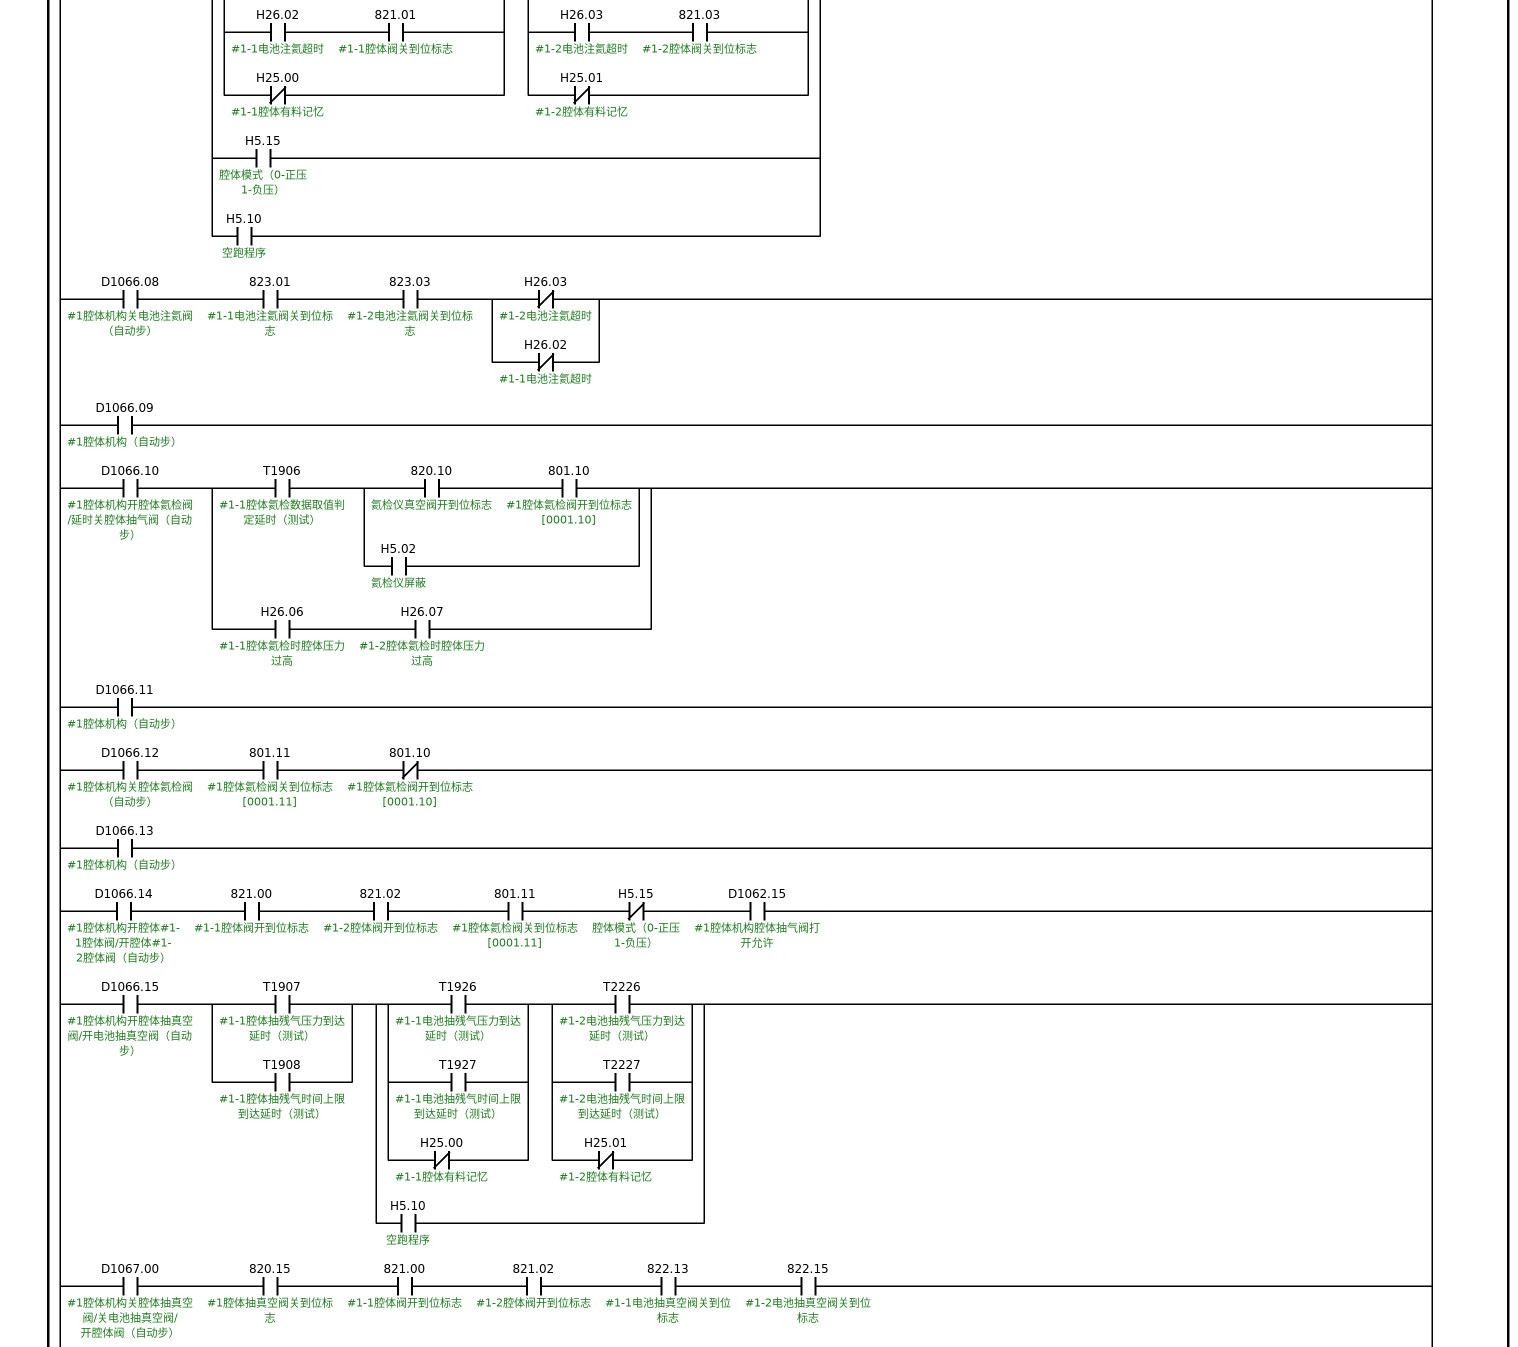
; [picture p192: 氦检机构 / 氦检腔1自动, rungs 7-7]

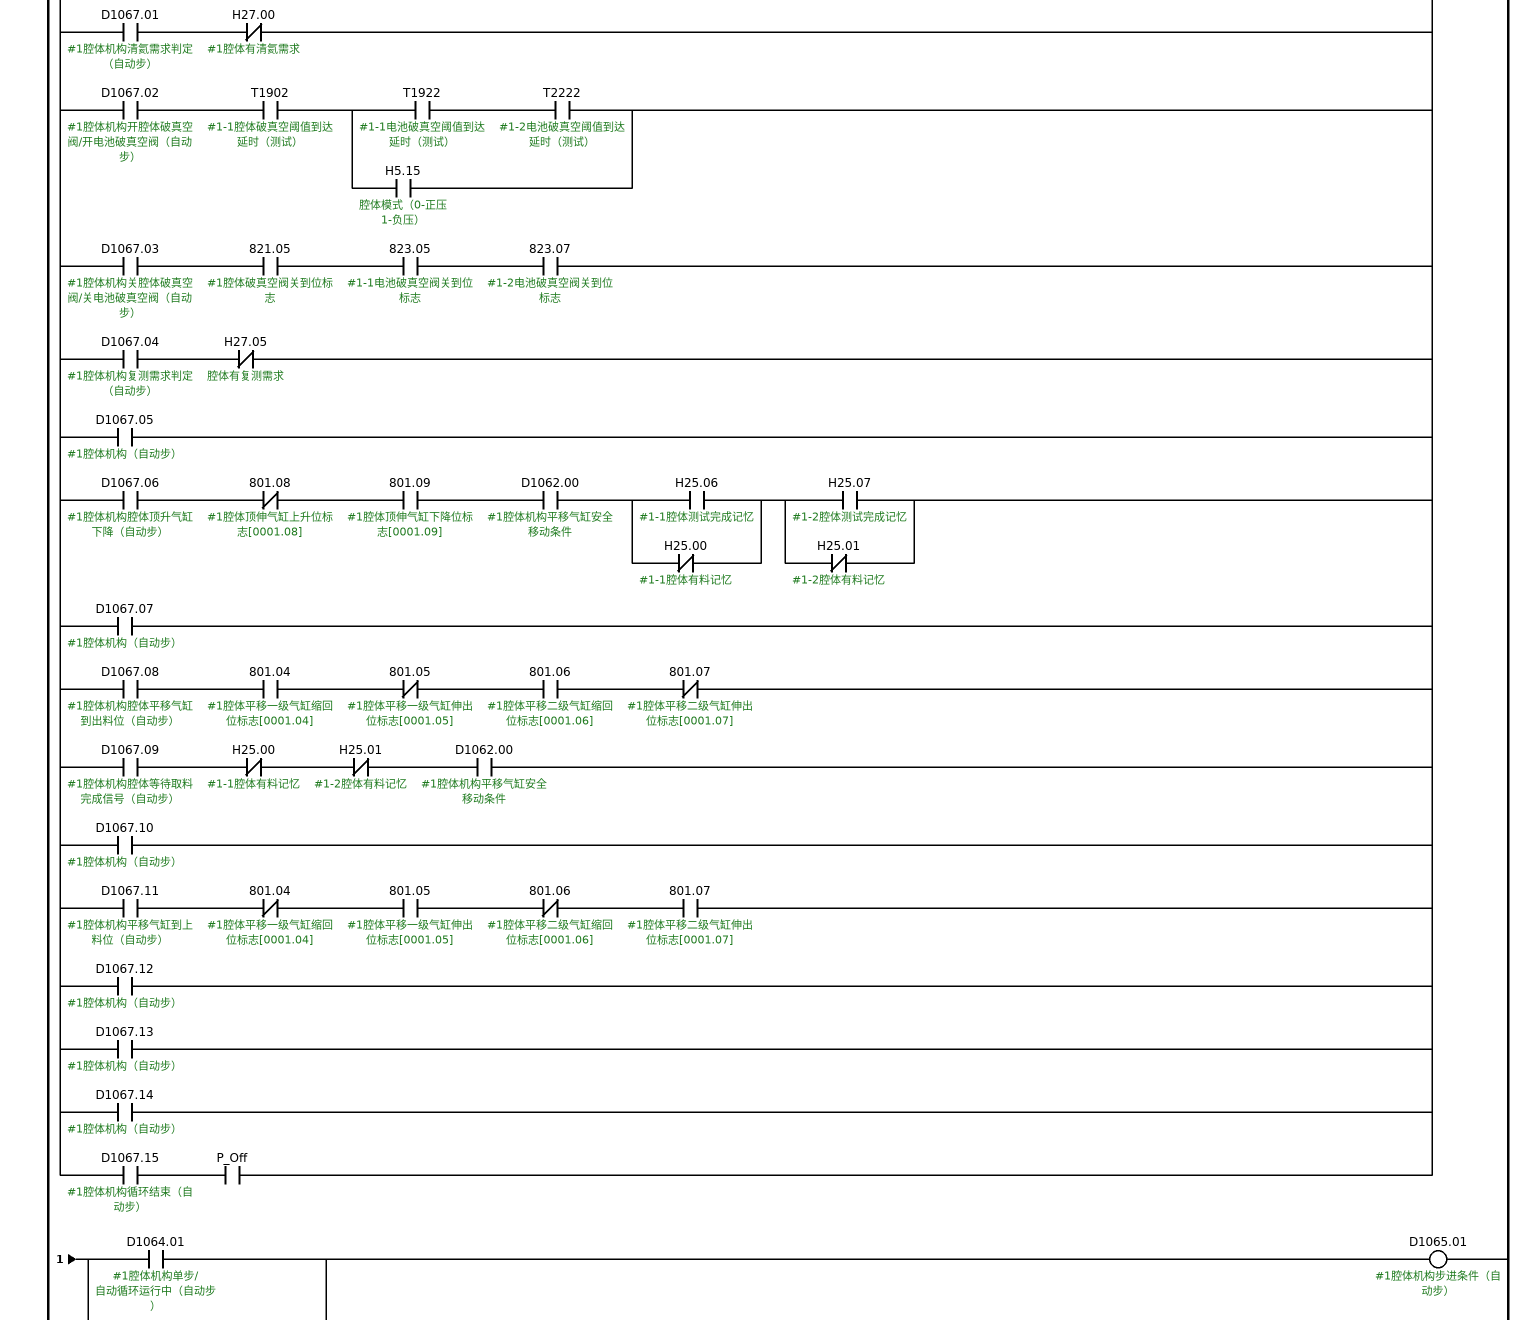

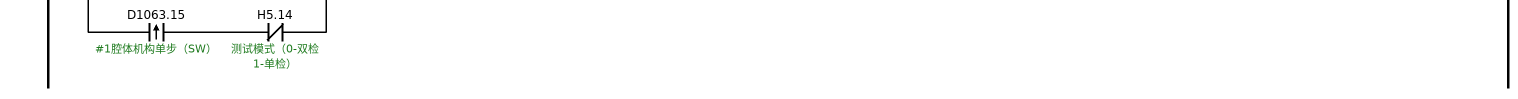
; rung 7: #1腔体机构步进条件（自动步）
LD D1066.00  ; #1腔体机构自动开始（自动步）
AND T1530  ; #1腔体机构开始运行条件延时(自动步)
LD D1066.01  ; #1腔体机构平移气缸到氦检位/数据初始化（自动步）
ANDNOT 801.04  ; #1腔体平移一级气缸缩回位标志[0001.04]
AND 801.05  ; #1腔体平移一级气缸伸出位标志[0001.05]
AND 801.06  ; #1腔体平移二级气缸缩回位标志[0001.06]
ANDNOT 801.07  ; #1腔体平移二级气缸伸出位标志[0001.07]
AND T1531  ; #1腔体机构数据初始化延时（自动步）
ORLD
LD D1066.02  ; #1腔体机构腔体顶升气缸上升（自动步）
AND 801.08  ; #1腔体顶伸气缸上升位标志[0001.08]
ANDNOT 801.09  ; #1腔体顶伸气缸下降位标志[0001.09]
ORLD
LD D1066.03  ; #1腔体机构等待氦检阀打开条件及腔体抽气阀打开条件/开腔体阀（自动步）
AND 821.00  ; #1-1腔体阀开到位标志
AND 821.02  ; #1-2腔体阀开到位标志
ANDNOT H32.00  ; #2腔体有清氦需求
ANDNOT H37.00  ; #3腔体有清氦需求
AND D1062.15  ; #1腔体机构腔体抽气阀打开允许
AND D1062.14  ; #1腔体氦检阀打开允许条件
LD W380.15  ; 氦检仪漏率低于设定值（稳态）
OR H5.02  ; 氦检仪屏蔽
ANDLD
AND=L(301) D1074 #0  ; #1腔体机构清氦步序号
ORLD
OR D1066.04  ; #1腔体机构（自动步）
LD D1066.05  ; #1腔体机构腔体抽气阀打开/延时开电池抽气阀（自动步）
LD T1900  ; #1-1腔体抽真空阈值到达延时（测试）
LD 822.12  ; #1-1电池抽真空阀开到位标志
AND T1920  ; #1-1电池抽真空阈值到达延时（测试）
LD H26.00  ; #1-1电池泄漏
ANDNOT H26.01  ; #1-2电池泄漏
ORLD
ORNOT H25.00  ; #1-1腔体有料记忆
LD 822.14  ; #1-2电池抽真空阀开到位标志
AND T2220  ; #1-2电池抽真空阈值到达延时（测试）
LDNOT H26.00  ; #1-1电池泄漏
AND H26.01  ; #1-2电池泄漏
ORLD
ORNOT H25.01  ; #1-2腔体有料记忆
ANDLD
OR H5.15  ; 腔体模式（0-正压 1-负压）
OR H5.10  ; 空跑程序
ANDLD
LD H26.04  ; #1-1腔体抽真空NG
ORNOT H25.00  ; #1-1腔体有料记忆
LD H26.05  ; #1-2腔体抽真空NG
ORNOT H25.01  ; #1-2腔体有料记忆
ANDLD
ORLD
LD H26.00  ; #1-1电池泄漏
AND H26.01  ; #1-2电池泄漏
ORLD
ANDLD
ORLD
LD D1066.06  ; #1腔体机构关电池抽气阀（自动步）  // 单个电池出现电池泄漏时，需将对应的腔体阀门关闭
ANDNOT W407.14  ; 设备氦气压力信号[alm]
ANDNOT W407.15  ; 精密调压阀信号[alm]
AND 822.13  ; #1-1电池抽真空阀关到位标志
AND 822.15  ; #1-2电池抽真空阀关到位标志
ANDNOT H26.04  ; #1-1腔体抽真空NG
ANDNOT H26.05  ; #1-2腔体抽真空NG
LD H26.00  ; #1-1电池泄漏
AND 821.01  ; #1-1腔体阀关到位标志
ORNOT H26.00  ; #1-1电池泄漏
ORNOT H25.00  ; #1-1腔体有料记忆
ANDLD
LD H26.01  ; #1-2电池泄漏
AND 821.03  ; #1-2腔体阀关到位标志
ORNOT H26.01  ; #1-2电池泄漏
ORNOT H25.01  ; #1-2腔体有料记忆
ANDLD
ORLD
LD D1066.07  ; #1腔体机构开电池注氦阀（自动步）  // 单个电池出现注氦超时时，需将对应的腔体阀门关闭
LD 823.00  ; #1-1电池注氦阀开到位标志
AND T1924  ; #1-1电池注氦压力到达延时（测试）
OR H26.00  ; #1-1电池泄漏
LD H26.02  ; #1-1电池注氦超时
AND 821.01  ; #1-1腔体阀关到位标志
ORLD
ORNOT H25.00  ; #1-1腔体有料记忆
LD 823.02  ; #1-2电池注氦阀开到位标志
AND T2224  ; #1-2电池注氦压力到达延时（测试）
OR H26.01  ; #1-2电池泄漏
LD H26.03  ; #1-2电池注氦超时
AND 821.03  ; #1-2腔体阀关到位标志
ORLD
ORNOT H25.01  ; #1-2腔体有料记忆
ANDLD
OR H5.15  ; 腔体模式（0-正压 1-负压）
OR H5.10  ; 空跑程序
ANDLD
ORLD
LD D1066.08  ; #1腔体机构关电池注氦阀（自动步）
AND 823.01  ; #1-1电池注氦阀关到位标志
AND 823.03  ; #1-2电池注氦阀关到位标志
LDNOT H26.03  ; #1-2电池注氦超时
ORNOT H26.02  ; #1-1电池注氦超时
ANDLD
ORLD
OR D1066.09  ; #1腔体机构（自动步）
LD D1066.10  ; #1腔体机构开腔体氦检阀/延时关腔体抽气阀（自动步）
LD T1906  ; #1-1腔体氦检数据取值判定延时（测试）
LD 820.10  ; 氦检仪真空阀开到位标志
AND 801.10  ; #1腔体氦检阀开到位标志[0001.10]
OR H5.02  ; 氦检仪屏蔽
ANDLD
LD H26.06  ; #1-1腔体氦检时腔体压力过高
AND H26.07  ; #1-2腔体氦检时腔体压力过高
ORLD
ANDLD
ORLD
OR D1066.11  ; #1腔体机构（自动步）
LD D1066.12  ; #1腔体机构关腔体氦检阀（自动步）
AND 801.11  ; #1腔体氦检阀关到位标志[0001.11]
ANDNOT 801.10  ; #1腔体氦检阀开到位标志[0001.10]
ORLD
OR D1066.13  ; #1腔体机构（自动步）
LD D1066.14  ; #1腔体机构开腔体#1-1腔体阀/开腔体#1-2腔体阀（自动步）
AND 821.00  ; #1-1腔体阀开到位标志
AND 821.02  ; #1-2腔体阀开到位标志
AND 801.11  ; #1腔体氦检阀关到位标志[0001.11]
ANDNOT H5.15  ; 腔体模式（0-正压 1-负压）
AND D1062.15  ; #1腔体机构腔体抽气阀打开允许
ORLD
LD D1066.15  ; #1腔体机构开腔体抽真空阀/开电池抽真空阀（自动步）
LD T1907  ; #1-1腔体抽残气压力到达延时（测试）
OR T1908  ; #1-1腔体抽残气时间上限到达延时（测试）
ANDLD
LD T1926  ; #1-1电池抽残气压力到达延时（测试）
OR T1927  ; #1-1电池抽残气时间上限到达延时（测试）
ORNOT H25.00  ; #1-1腔体有料记忆
LD T2226  ; #1-2电池抽残气压力到达延时（测试）
OR T2227  ; #1-2电池抽残气时间上限到达延时（测试）
ORNOT H25.01  ; #1-2腔体有料记忆
ANDLD
OR H5.10  ; 空跑程序
ANDLD
ORLD
LD D1067.00  ; #1腔体机构关腔体抽真空阀/关电池抽真空阀/开腔体阀（自动步）
AND 820.15  ; #1腔体抽真空阀关到位标志
AND 821.00  ; #1-1腔体阀开到位标志
AND 821.02  ; #1-2腔体阀开到位标志
AND 822.13  ; #1-1电池抽真空阀关到位标志
AND 822.15  ; #1-2电池抽真空阀关到位标志
ORLD
LD D1067.01  ; #1腔体机构清氦需求判定（自动步）
ANDNOT H27.00  ; #1腔体有清氦需求
ORLD
LD D1067.02  ; #1腔体机构开腔体破真空阀/开电池破真空阀（自动步）
AND T1902  ; #1-1腔体破真空阈值到达延时（测试）
LD T1922  ; #1-1电池破真空阈值到达延时（测试）
AND T2222  ; #1-2电池破真空阈值到达延时（测试）
OR H5.15  ; 腔体模式（0-正压 1-负压）
ANDLD
ORLD
LD D1067.03  ; #1腔体机构关腔体破真空阀/关电池破真空阀（自动步）
AND 821.05  ; #1腔体破真空阀关到位标志
AND 823.05  ; #1-1电池破真空阀关到位标志
AND 823.07  ; #1-2电池破真空阀关到位标志
ORLD
LD D1067.04  ; #1腔体机构复测需求判定（自动步）
ANDNOT H27.05  ; 腔体有复测需求
ORLD
OR D1067.05  ; #1腔体机构（自动步）
LD D1067.06  ; #1腔体机构腔体顶升气缸下降（自动步）
ANDNOT 801.08  ; #1腔体顶伸气缸上升位标志[0001.08]
AND 801.09  ; #1腔体顶伸气缸下降位标志[0001.09]
AND D1062.00  ; #1腔体机构平移气缸安全移动条件
LD H25.06  ; #1-1腔体测试完成记忆
ORNOT H25.00  ; #1-1腔体有料记忆
ANDLD
LD H25.07  ; #1-2腔体测试完成记忆
ORNOT H25.01  ; #1-2腔体有料记忆
ANDLD
ORLD
OR D1067.07  ; #1腔体机构（自动步）
LD D1067.08  ; #1腔体机构腔体平移气缸到出料位（自动步）
AND 801.04  ; #1腔体平移一级气缸缩回位标志[0001.04]
ANDNOT 801.05  ; #1腔体平移一级气缸伸出位标志[0001.05]
AND 801.06  ; #1腔体平移二级气缸缩回位标志[0001.06]
ANDNOT 801.07  ; #1腔体平移二级气缸伸出位标志[0001.07]
ORLD
LD D1067.09  ; #1腔体机构腔体等待取料完成信号（自动步）
ANDNOT H25.00  ; #1-1腔体有料记忆
ANDNOT H25.01  ; #1-2腔体有料记忆
AND D1062.00  ; #1腔体机构平移气缸安全移动条件
ORLD
OR D1067.10  ; #1腔体机构（自动步）
LD D1067.11  ; #1腔体机构平移气缸到上料位（自动步）
ANDNOT 801.04  ; #1腔体平移一级气缸缩回位标志[0001.04]
AND 801.05  ; #1腔体平移一级气缸伸出位标志[0001.05]
ANDNOT 801.06  ; #1腔体平移二级气缸缩回位标志[0001.06]
AND 801.07  ; #1腔体平移二级气缸伸出位标志[0001.07]
ORLD
OR D1067.12  ; #1腔体机构（自动步）
OR D1067.13  ; #1腔体机构（自动步）
OR D1067.14  ; #1腔体机构（自动步）
LD D1067.15  ; #1腔体机构循环结束（自动步）
AND P_Off
ORLD
LD D1064.01  ; #1腔体机构单步/自动循环运行中（自动步）
@LD D1063.15  ; #1腔体机构单步（SW）
ANDNOT H5.14  ; 测试模式（0-双检 1-单检）
ORLD
ANDLD
OUT D1065.01  ; #1腔体机构步进条件（自动步）

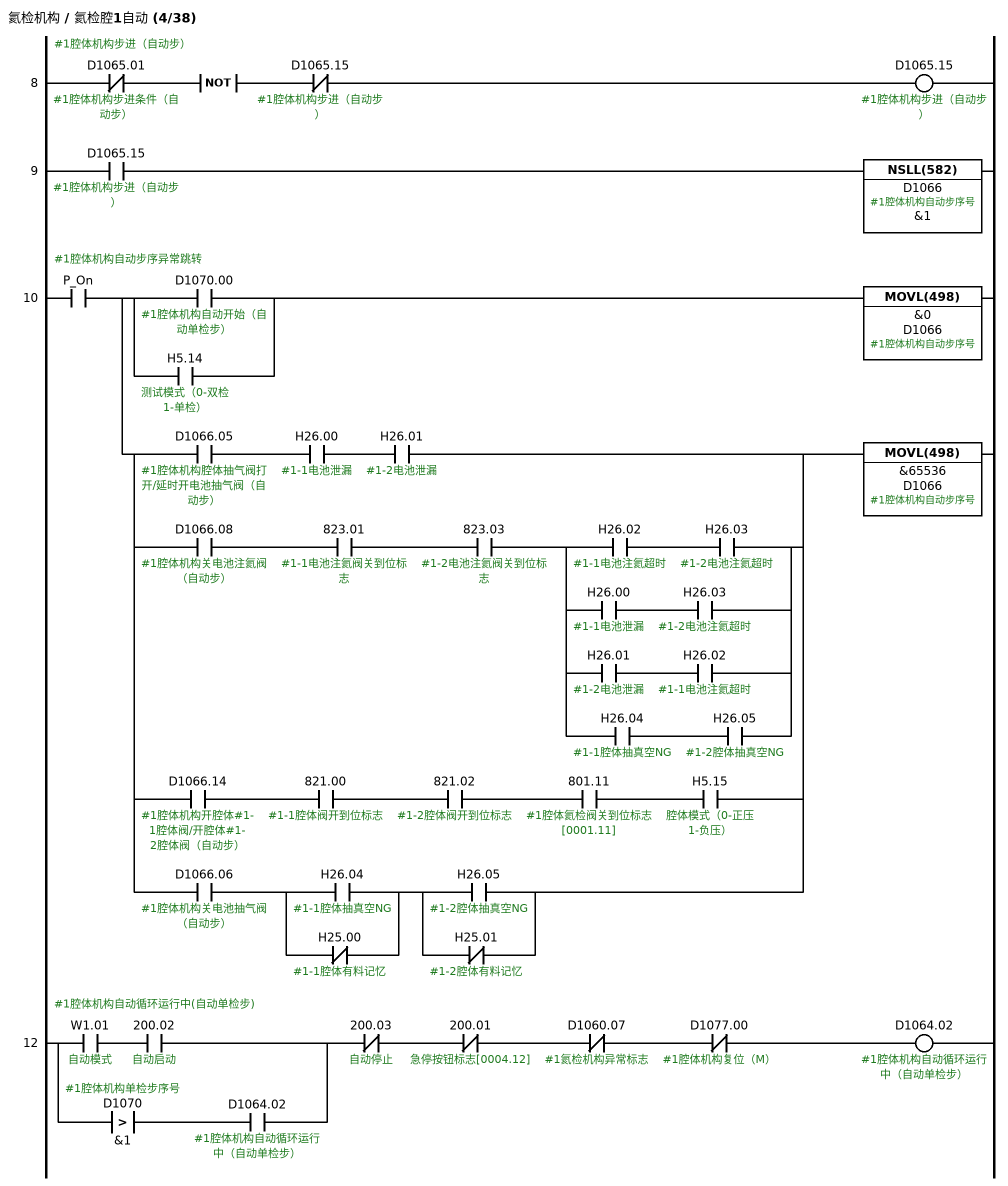
; rung 8: #1腔体机构步进（自动步）
LDNOT D1065.01  ; #1腔体机构步进条件（自动步）
NOT(520)
ANDNOT D1065.15  ; #1腔体机构步进（自动步）
OUT D1065.15  ; #1腔体机构步进（自动步）
; rung 9
LD D1065.15  ; #1腔体机构步进（自动步）
NSLL(582) D1066 &1  ; #1腔体机构自动步序号
; rung 10: #1腔体机构自动步序异常跳转
LD P_On
OUT TR0
LD D1070.00  ; #1腔体机构自动开始（自动单检步）
OR H5.14  ; 测试模式（0-双检 1-单检）
ANDLD
MOVL(498) &0 D1066  ; #1腔体机构自动步序号  // 测试模式为单检模式，腔体进入到复测步序时，将腔体机构自动步序清零
LD TR0
LD D1066.05  ; #1腔体机构腔体抽气阀打开/延时开电池抽气阀（自动步）
AND H26.00  ; #1-1电池泄漏
AND H26.01  ; #1-2电池泄漏
LD D1066.08  ; #1腔体机构关电池注氦阀（自动步）
AND 823.01  ; #1-1电池注氦阀关到位标志
AND 823.03  ; #1-2电池注氦阀关到位标志
LD H26.02  ; #1-1电池注氦超时
AND H26.03  ; #1-2电池注氦超时
LD H26.00  ; #1-1电池泄漏
AND H26.03  ; #1-2电池注氦超时
ORLD
LD H26.01  ; #1-2电池泄漏
AND H26.02  ; #1-1电池注氦超时
ORLD
LD H26.04  ; #1-1腔体抽真空NG
AND H26.05  ; #1-2腔体抽真空NG
ORLD
ANDLD
ORLD
LD D1066.14  ; #1腔体机构开腔体#1-1腔体阀/开腔体#1-2腔体阀（自动步）  // 负压模式不需要进行氦检后抽真空动作
AND 821.00  ; #1-1腔体阀开到位标志
AND 821.02  ; #1-2腔体阀开到位标志
AND 801.11  ; #1腔体氦检阀关到位标志[0001.11]
AND H5.15  ; 腔体模式（0-正压 1-负压）
ORLD
LD D1066.06  ; #1腔体机构关电池抽气阀（自动步）
LD H26.04  ; #1-1腔体抽真空NG
ORNOT H25.00  ; #1-1腔体有料记忆
ANDLD
LD H26.05  ; #1-2腔体抽真空NG
ORNOT H25.01  ; #1-2腔体有料记忆
ANDLD
ORLD
ANDLD
MOVL(498) &65536 D1066  ; #1腔体机构自动步序号  // 出现腔体抽真空NG，双电池抽真空NG，双电池注氦超时的情况，均跳转至自动步序D1067.0
; rung 11: ******************************* / 自动单检步序 / *******************************
; rung 12: #1腔体机构自动循环运行中(自动单检步)
LD W1.01  ; 自动模式
AND 200.02  ; 自动启动
LD>L(321) D1070 &1  ; #1腔体机构单检步序号
AND D1064.02  ; #1腔体机构自动循环运行中（自动单检步）
ORLD
ANDNOT 200.03  ; 自动停止
ANDNOT 200.01  ; 急停按钮标志[0004.12]
ANDNOT D1060.07  ; #1氦检机构异常标志
ANDNOT D1077.00  ; #1腔体机构复位（M）
OUT D1064.02  ; #1腔体机构自动循环运行中（自动单检步）

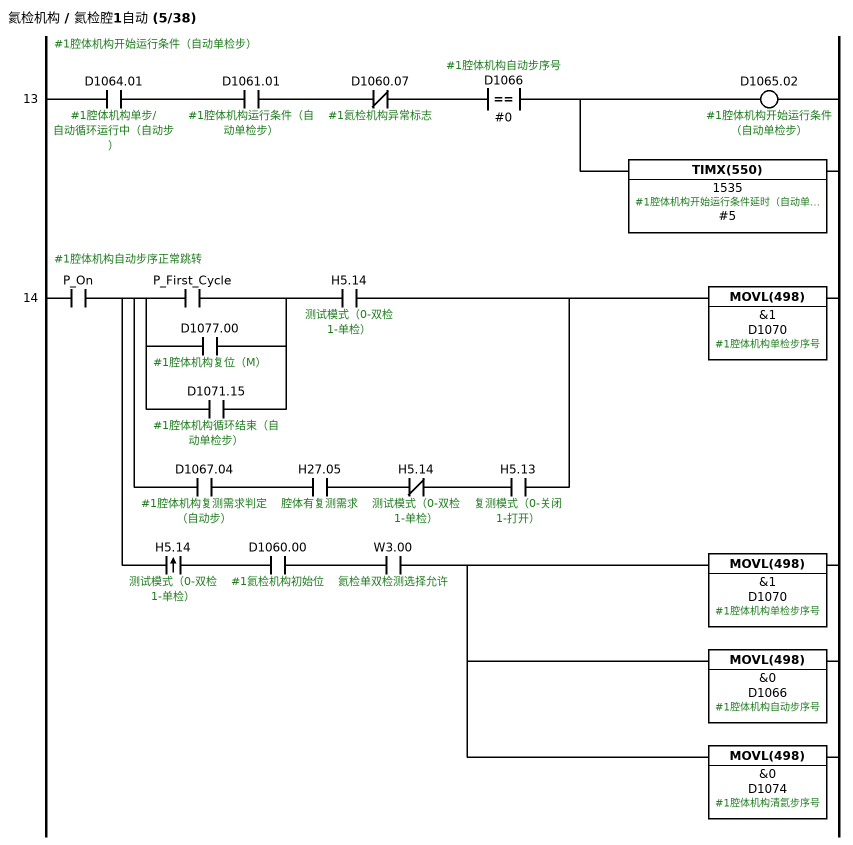
; rung 13: #1腔体机构开始运行条件（自动单检步）
LD D1064.01  ; #1腔体机构单步/自动循环运行中（自动步）
AND D1061.01  ; #1腔体机构运行条件（自动单检步）
ANDNOT D1060.07  ; #1氦检机构异常标志
AND=L(301) D1066 #0  ; #1腔体机构自动步序号
OUT D1065.02  ; #1腔体机构开始运行条件（自动单检步）
TIMX(550) 1535 #5  ; #1腔体机构开始运行条件延时（自动单检步）
; rung 14: #1腔体机构自动步序正常跳转
LD P_On
OUT TR0
LD P_First_Cycle
OR D1077.00  ; #1腔体机构复位（M）
OR D1071.15  ; #1腔体机构循环结束（自动单检步）
AND H5.14  ; 测试模式（0-双检 1-单检）
LD D1067.04  ; #1腔体机构复测需求判定（自动步）
AND H27.05  ; 腔体有复测需求
ANDNOT H5.14  ; 测试模式（0-双检 1-单检）
AND H5.13  ; 复测模式（0-关闭 1-打开）
ORLD
ANDLD
MOVL(498) &1 D1070  ; #1腔体机构单检步序号
LD TR0
@AND H5.14  ; 测试模式（0-双检 1-单检）
AND D1060.00  ; #1氦检机构初始位
AND W3.00  ; 氦检单双检测选择允许
MOVL(498) &1 D1070  ; #1腔体机构单检步序号
MOVL(498) &0 D1066  ; #1腔体机构自动步序号
MOVL(498) &0 D1074  ; #1腔体机构清氦步序号

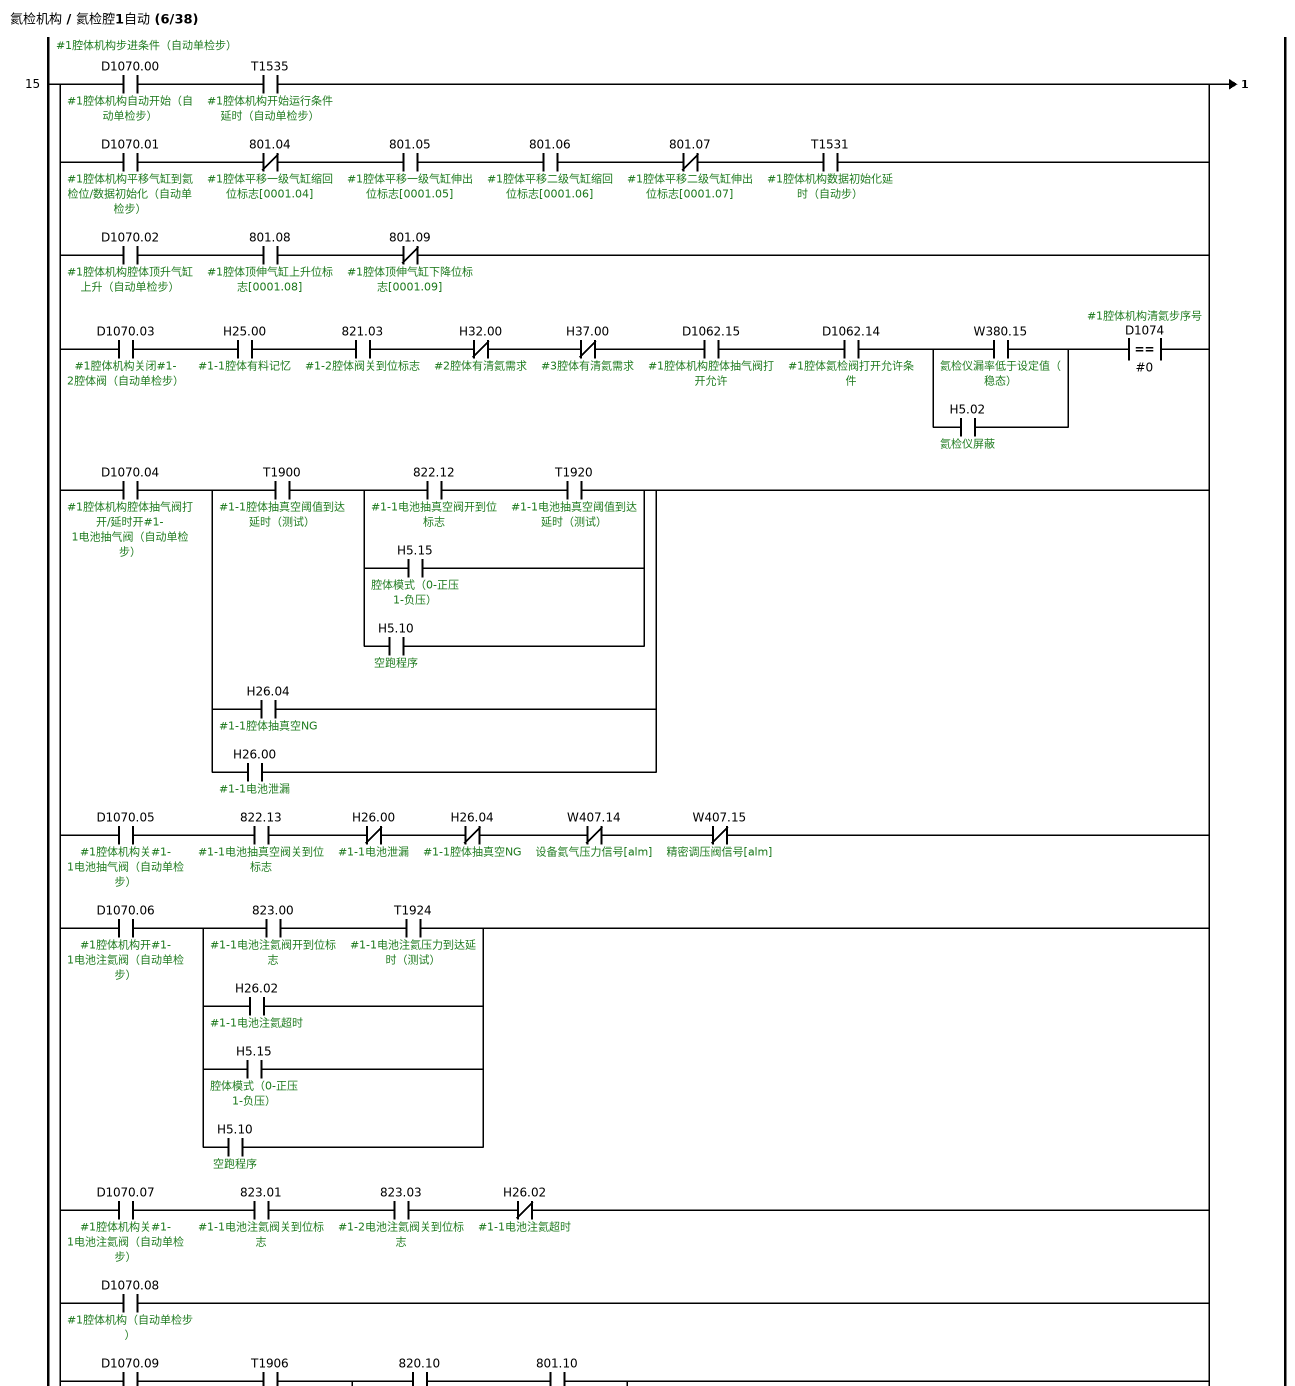

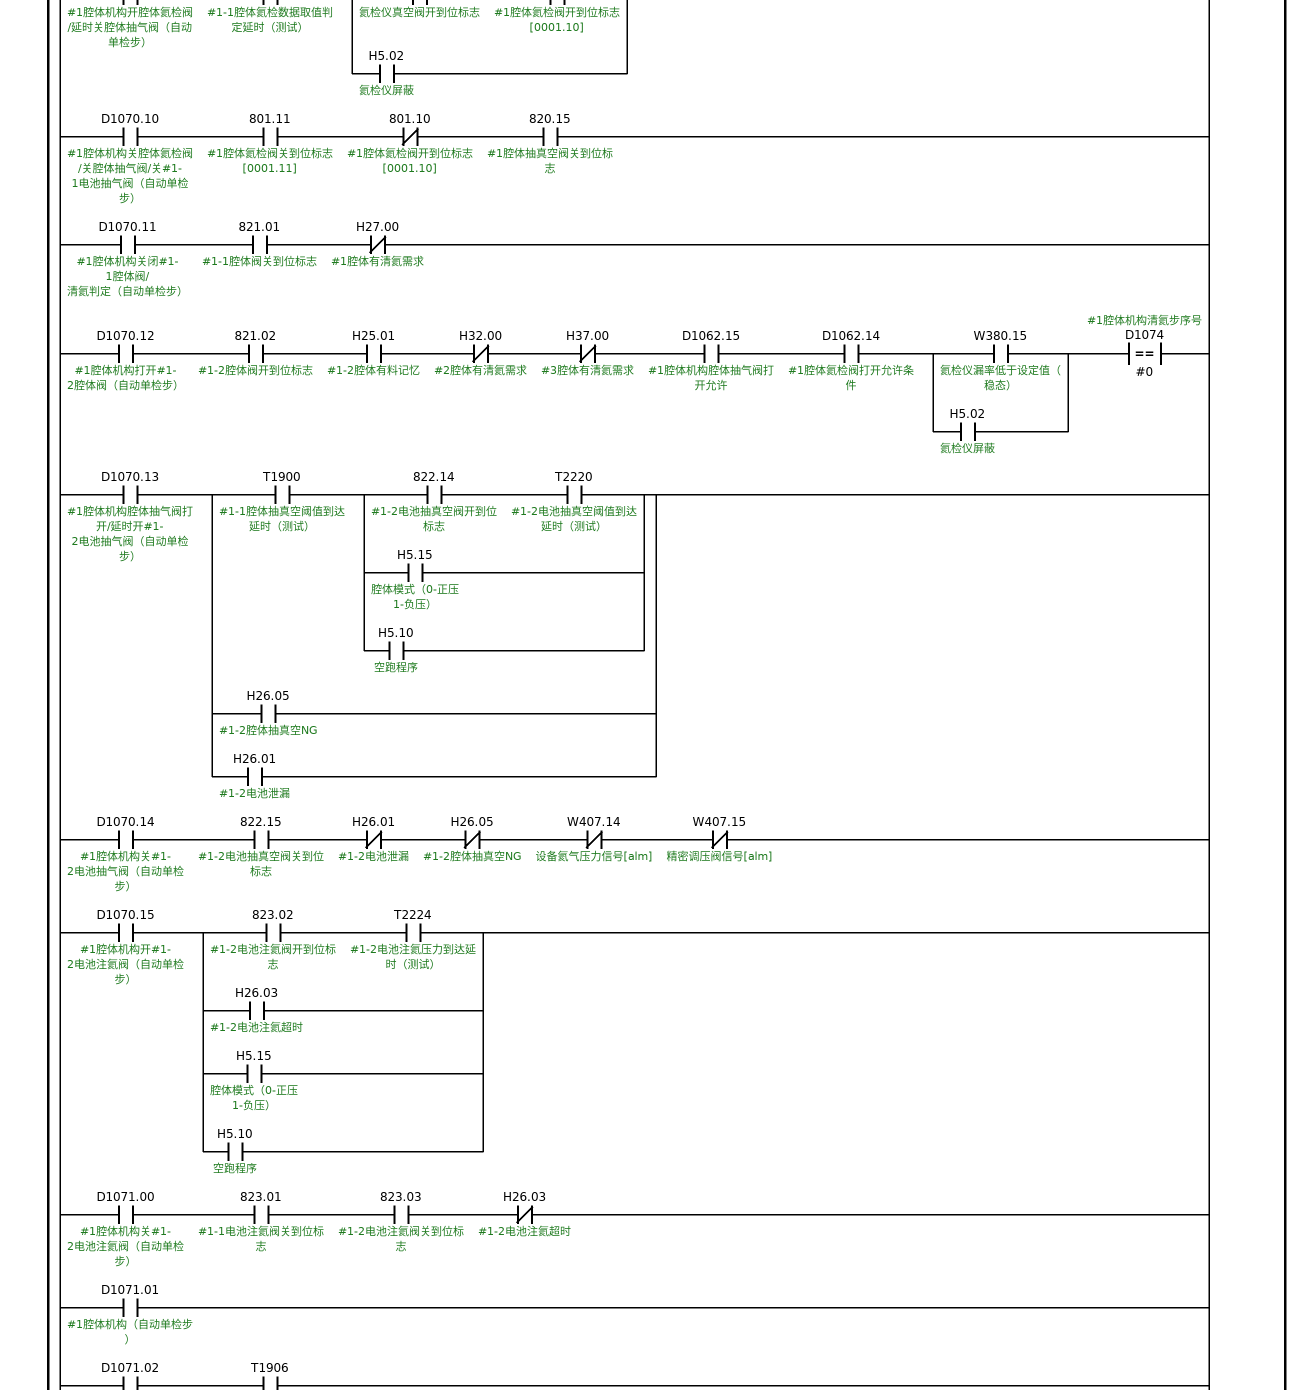

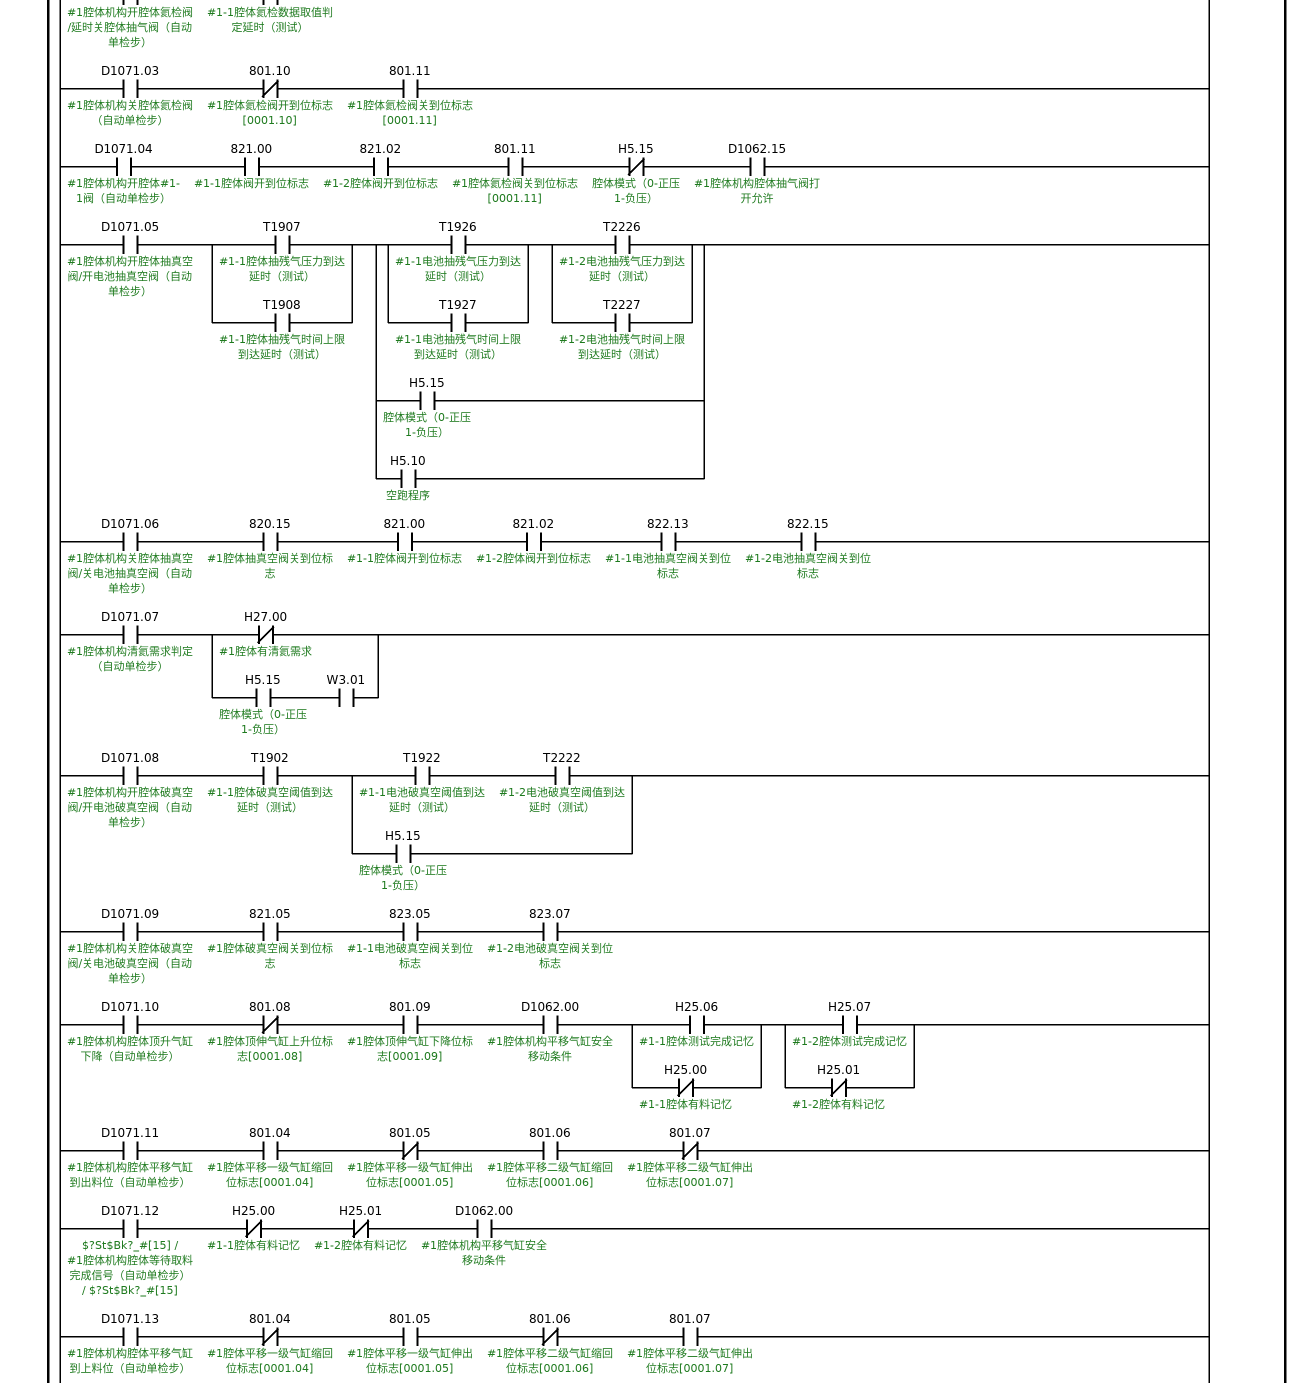

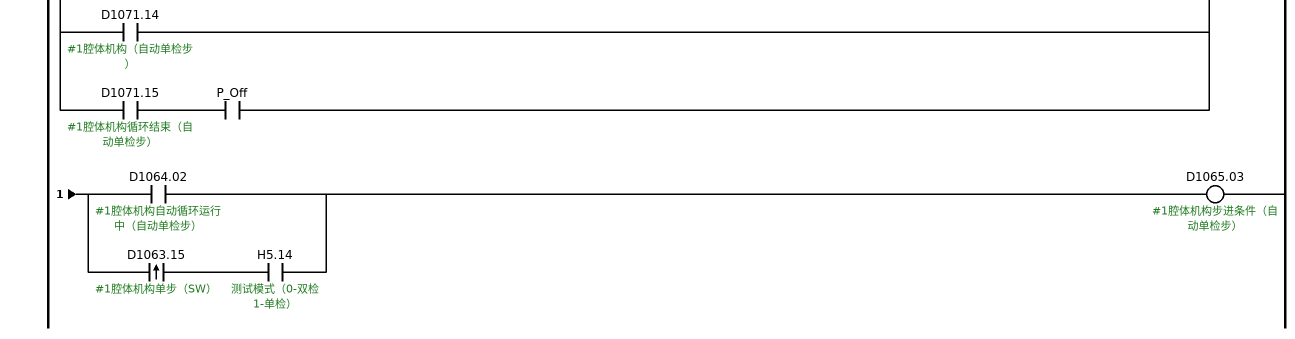
; rung 15: #1腔体机构步进条件（自动单检步）
LD D1070.00  ; #1腔体机构自动开始（自动单检步）
AND T1535  ; #1腔体机构开始运行条件延时（自动单检步）
LD D1070.01  ; #1腔体机构平移气缸到氦检位/数据初始化（自动单检步）
ANDNOT 801.04  ; #1腔体平移一级气缸缩回位标志[0001.04]
AND 801.05  ; #1腔体平移一级气缸伸出位标志[0001.05]
AND 801.06  ; #1腔体平移二级气缸缩回位标志[0001.06]
ANDNOT 801.07  ; #1腔体平移二级气缸伸出位标志[0001.07]
AND T1531  ; #1腔体机构数据初始化延时（自动步）
ORLD
LD D1070.02  ; #1腔体机构腔体顶升气缸上升（自动单检步）
AND 801.08  ; #1腔体顶伸气缸上升位标志[0001.08]
ANDNOT 801.09  ; #1腔体顶伸气缸下降位标志[0001.09]
ORLD
LD D1070.03  ; #1腔体机构关闭#1-2腔体阀（自动单检步）
AND H25.00  ; #1-1腔体有料记忆
AND 821.03  ; #1-2腔体阀关到位标志
ANDNOT H32.00  ; #2腔体有清氦需求
ANDNOT H37.00  ; #3腔体有清氦需求
AND D1062.15  ; #1腔体机构腔体抽气阀打开允许
AND D1062.14  ; #1腔体氦检阀打开允许条件
LD W380.15  ; 氦检仪漏率低于设定值（稳态）
OR H5.02  ; 氦检仪屏蔽
ANDLD
AND=L(301) D1074 #0  ; #1腔体机构清氦步序号
ORLD
LD D1070.04  ; #1腔体机构腔体抽气阀打开/延时开#1-1电池抽气阀（自动单检步）
LD T1900  ; #1-1腔体抽真空阈值到达延时（测试）
LD 822.12  ; #1-1电池抽真空阀开到位标志
AND T1920  ; #1-1电池抽真空阈值到达延时（测试）
OR H5.15  ; 腔体模式（0-正压 1-负压）
OR H5.10  ; 空跑程序
ANDLD
OR H26.04  ; #1-1腔体抽真空NG
OR H26.00  ; #1-1电池泄漏
ANDLD
ORLD
LD D1070.05  ; #1腔体机构关#1-1电池抽气阀（自动单检步）
AND 822.13  ; #1-1电池抽真空阀关到位标志
ANDNOT H26.00  ; #1-1电池泄漏
ANDNOT H26.04  ; #1-1腔体抽真空NG
ANDNOT W407.14  ; 设备氦气压力信号[alm]
ANDNOT W407.15  ; 精密调压阀信号[alm]
ORLD
LD D1070.06  ; #1腔体机构开#1-1电池注氦阀（自动单检步）
LD 823.00  ; #1-1电池注氦阀开到位标志
AND T1924  ; #1-1电池注氦压力到达延时（测试）
OR H26.02  ; #1-1电池注氦超时
OR H5.15  ; 腔体模式（0-正压 1-负压）
OR H5.10  ; 空跑程序
ANDLD
ORLD
LD D1070.07  ; #1腔体机构关#1-1电池注氦阀（自动单检步）
AND 823.01  ; #1-1电池注氦阀关到位标志
AND 823.03  ; #1-2电池注氦阀关到位标志
ANDNOT H26.02  ; #1-1电池注氦超时
ORLD
OR D1070.08  ; #1腔体机构（自动单检步）
LD D1070.09  ; #1腔体机构开腔体氦检阀/延时关腔体抽气阀（自动单检步）
AND T1906  ; #1-1腔体氦检数据取值判定延时（测试）
LD 820.10  ; 氦检仪真空阀开到位标志
AND 801.10  ; #1腔体氦检阀开到位标志[0001.10]
OR H5.02  ; 氦检仪屏蔽
ANDLD
ORLD
LD D1070.10  ; #1腔体机构关腔体氦检阀/关腔体抽气阀/关#1-1电池抽气阀（自动单检步）
AND 801.11  ; #1腔体氦检阀关到位标志[0001.11]
ANDNOT 801.10  ; #1腔体氦检阀开到位标志[0001.10]
AND 820.15  ; #1腔体抽真空阀关到位标志
ORLD
LD D1070.11  ; #1腔体机构关闭#1-1腔体阀/清氦判定（自动单检步）
AND 821.01  ; #1-1腔体阀关到位标志
ANDNOT H27.00  ; #1腔体有清氦需求
ORLD
LD D1070.12  ; #1腔体机构打开#1-2腔体阀（自动单检步）
AND 821.02  ; #1-2腔体阀开到位标志
AND H25.01  ; #1-2腔体有料记忆
ANDNOT H32.00  ; #2腔体有清氦需求
ANDNOT H37.00  ; #3腔体有清氦需求
AND D1062.15  ; #1腔体机构腔体抽气阀打开允许
AND D1062.14  ; #1腔体氦检阀打开允许条件
LD W380.15  ; 氦检仪漏率低于设定值（稳态）
OR H5.02  ; 氦检仪屏蔽
ANDLD
AND=L(301) D1074 #0  ; #1腔体机构清氦步序号
ORLD
LD D1070.13  ; #1腔体机构腔体抽气阀打开/延时开#1-2电池抽气阀（自动单检步）
LD T1900  ; #1-1腔体抽真空阈值到达延时（测试）
LD 822.14  ; #1-2电池抽真空阀开到位标志
AND T2220  ; #1-2电池抽真空阈值到达延时（测试）
OR H5.15  ; 腔体模式（0-正压 1-负压）
OR H5.10  ; 空跑程序
ANDLD
OR H26.05  ; #1-2腔体抽真空NG
OR H26.01  ; #1-2电池泄漏
ANDLD
ORLD
LD D1070.14  ; #1腔体机构关#1-2电池抽气阀（自动单检步）
AND 822.15  ; #1-2电池抽真空阀关到位标志
ANDNOT H26.01  ; #1-2电池泄漏
ANDNOT H26.05  ; #1-2腔体抽真空NG
ANDNOT W407.14  ; 设备氦气压力信号[alm]
ANDNOT W407.15  ; 精密调压阀信号[alm]
ORLD
LD D1070.15  ; #1腔体机构开#1-2电池注氦阀（自动单检步）
LD 823.02  ; #1-2电池注氦阀开到位标志
AND T2224  ; #1-2电池注氦压力到达延时（测试）
OR H26.03  ; #1-2电池注氦超时
OR H5.15  ; 腔体模式（0-正压 1-负压）
OR H5.10  ; 空跑程序
ANDLD
ORLD
LD D1071.00  ; #1腔体机构关#1-2电池注氦阀（自动单检步）
AND 823.01  ; #1-1电池注氦阀关到位标志
AND 823.03  ; #1-2电池注氦阀关到位标志
ANDNOT H26.03  ; #1-2电池注氦超时
ORLD
OR D1071.01  ; #1腔体机构（自动单检步）
LD D1071.02  ; #1腔体机构开腔体氦检阀/延时关腔体抽气阀（自动单检步）
AND T1906  ; #1-1腔体氦检数据取值判定延时（测试）
ORLD
LD D1071.03  ; #1腔体机构关腔体氦检阀（自动单检步）
ANDNOT 801.10  ; #1腔体氦检阀开到位标志[0001.10]
AND 801.11  ; #1腔体氦检阀关到位标志[0001.11]
ORLD
LD D1071.04  ; #1腔体机构开腔体#1-1阀（自动单检步）
AND 821.00  ; #1-1腔体阀开到位标志
AND 821.02  ; #1-2腔体阀开到位标志
AND 801.11  ; #1腔体氦检阀关到位标志[0001.11]
ANDNOT H5.15  ; 腔体模式（0-正压 1-负压）
AND D1062.15  ; #1腔体机构腔体抽气阀打开允许
ORLD
LD D1071.05  ; #1腔体机构开腔体抽真空阀/开电池抽真空阀（自动单检步）
LD T1907  ; #1-1腔体抽残气压力到达延时（测试）
OR T1908  ; #1-1腔体抽残气时间上限到达延时（测试）
ANDLD
LD T1926  ; #1-1电池抽残气压力到达延时（测试）
OR T1927  ; #1-1电池抽残气时间上限到达延时（测试）
LD T2226  ; #1-2电池抽残气压力到达延时（测试）
OR T2227  ; #1-2电池抽残气时间上限到达延时（测试）
ANDLD
OR H5.15  ; 腔体模式（0-正压 1-负压）
OR H5.10  ; 空跑程序
ANDLD
ORLD
LD D1071.06  ; #1腔体机构关腔体抽真空阀/关电池抽真空阀（自动单检步）
AND 820.15  ; #1腔体抽真空阀关到位标志
AND 821.00  ; #1-1腔体阀开到位标志
AND 821.02  ; #1-2腔体阀开到位标志
AND 822.13  ; #1-1电池抽真空阀关到位标志
AND 822.15  ; #1-2电池抽真空阀关到位标志
ORLD
LD D1071.07  ; #1腔体机构清氦需求判定（自动单检步）
LDNOT H27.00  ; #1腔体有清氦需求
LD H5.15  ; 腔体模式（0-正压 1-负压）
AND W3.01
ORLD
ANDLD
ORLD
LD D1071.08  ; #1腔体机构开腔体破真空阀/开电池破真空阀（自动单检步）
AND T1902  ; #1-1腔体破真空阈值到达延时（测试）
LD T1922  ; #1-1电池破真空阈值到达延时（测试）
AND T2222  ; #1-2电池破真空阈值到达延时（测试）
OR H5.15  ; 腔体模式（0-正压 1-负压）
ANDLD
ORLD
LD D1071.09  ; #1腔体机构关腔体破真空阀/关电池破真空阀（自动单检步）
AND 821.05  ; #1腔体破真空阀关到位标志
AND 823.05  ; #1-1电池破真空阀关到位标志
AND 823.07  ; #1-2电池破真空阀关到位标志
ORLD
LD D1071.10  ; #1腔体机构腔体顶升气缸下降（自动单检步）
ANDNOT 801.08  ; #1腔体顶伸气缸上升位标志[0001.08]
AND 801.09  ; #1腔体顶伸气缸下降位标志[0001.09]
AND D1062.00  ; #1腔体机构平移气缸安全移动条件
LD H25.06  ; #1-1腔体测试完成记忆
ORNOT H25.00  ; #1-1腔体有料记忆
ANDLD
LD H25.07  ; #1-2腔体测试完成记忆
ORNOT H25.01  ; #1-2腔体有料记忆
ANDLD
ORLD
LD D1071.11  ; #1腔体机构腔体平移气缸到出料位（自动单检步）
AND 801.04  ; #1腔体平移一级气缸缩回位标志[0001.04]
ANDNOT 801.05  ; #1腔体平移一级气缸伸出位标志[0001.05]
AND 801.06  ; #1腔体平移二级气缸缩回位标志[0001.06]
ANDNOT 801.07  ; #1腔体平移二级气缸伸出位标志[0001.07]
ORLD
LD D1071.12  ; $?St$Bk?_#[15] / #1腔体机构腔体等待取料完成信号（自动单检步） / $?St$Bk?_#[15]
ANDNOT H25.00  ; #1-1腔体有料记忆
ANDNOT H25.01  ; #1-2腔体有料记忆
AND D1062.00  ; #1腔体机构平移气缸安全移动条件
ORLD
LD D1071.13  ; #1腔体机构腔体平移气缸到上料位（自动单检步）
ANDNOT 801.04  ; #1腔体平移一级气缸缩回位标志[0001.04]
AND 801.05  ; #1腔体平移一级气缸伸出位标志[0001.05]
ANDNOT 801.06  ; #1腔体平移二级气缸缩回位标志[0001.06]
AND 801.07  ; #1腔体平移二级气缸伸出位标志[0001.07]
ORLD
OR D1071.14  ; #1腔体机构（自动单检步）
LD D1071.15  ; #1腔体机构循环结束（自动单检步）
AND P_Off
ORLD
LD D1064.02  ; #1腔体机构自动循环运行中（自动单检步）
@LD D1063.15  ; #1腔体机构单步（SW）
AND H5.14  ; 测试模式（0-双检 1-单检）
ORLD
ANDLD
OUT D1065.03  ; #1腔体机构步进条件（自动单检步）

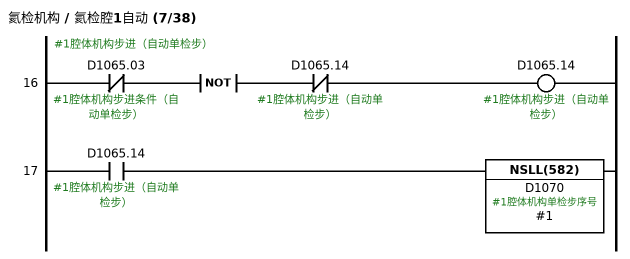
; rung 16: #1腔体机构步进（自动单检步）
LDNOT D1065.03  ; #1腔体机构步进条件（自动单检步）
NOT(520)
ANDNOT D1065.14  ; #1腔体机构步进（自动单检步）
OUT D1065.14  ; #1腔体机构步进（自动单检步）
; rung 17
LD D1065.14  ; #1腔体机构步进（自动单检步）
NSLL(582) D1070 #1  ; #1腔体机构单检步序号

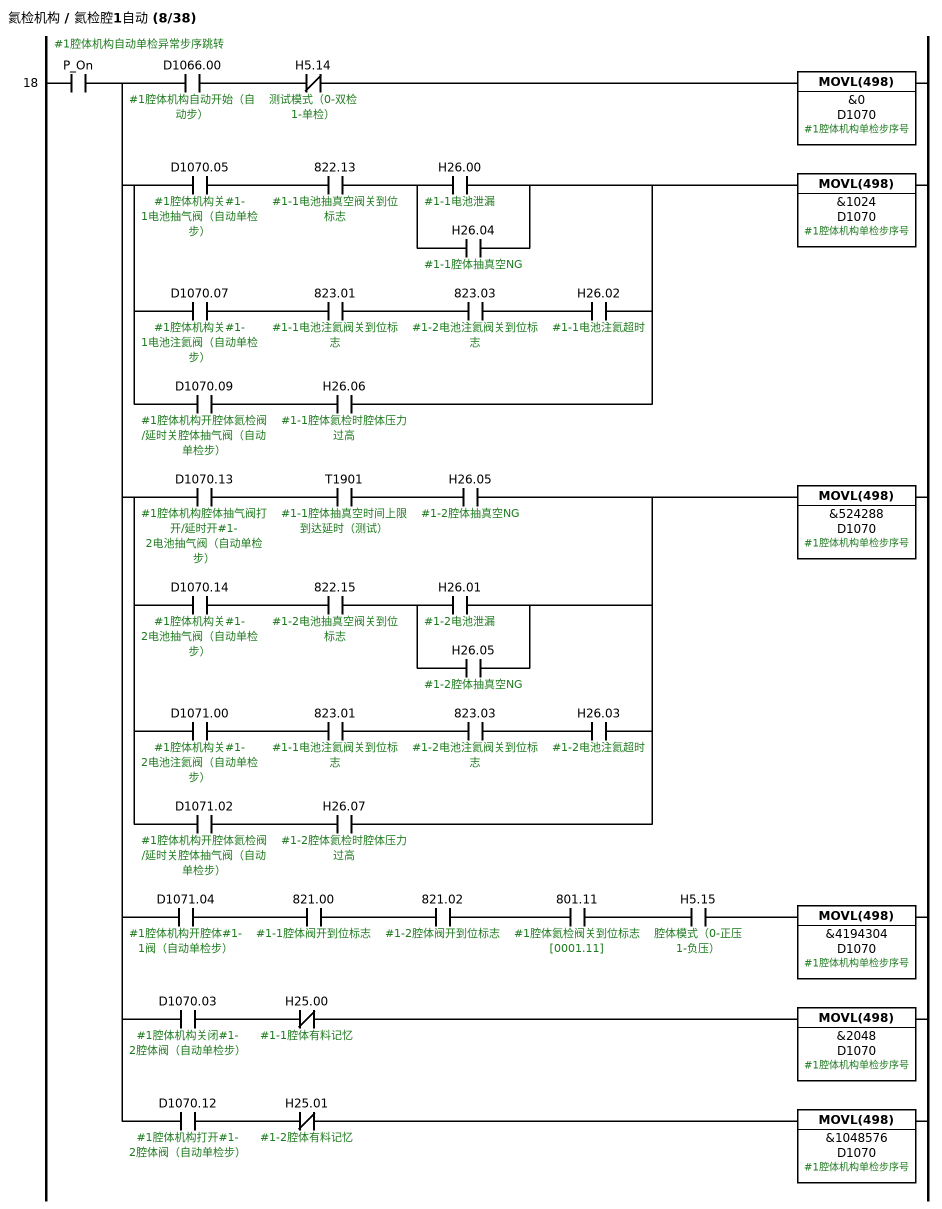
; rung 18: #1腔体机构自动单检异常步序跳转
LD P_On
OUT TR0
AND D1066.00  ; #1腔体机构自动开始（自动步）
ANDNOT H5.14  ; 测试模式（0-双检 1-单检）
MOVL(498) &0 D1070  ; #1腔体机构单检步序号
LD TR0
LD D1070.05  ; #1腔体机构关#1-1电池抽气阀（自动单检步）
AND 822.13  ; #1-1电池抽真空阀关到位标志
LD H26.00  ; #1-1电池泄漏
OR H26.04  ; #1-1腔体抽真空NG
ANDLD
LD D1070.07  ; #1腔体机构关#1-1电池注氦阀（自动单检步）
AND 823.01  ; #1-1电池注氦阀关到位标志
AND 823.03  ; #1-2电池注氦阀关到位标志
AND H26.02  ; #1-1电池注氦超时
ORLD
LD D1070.09  ; #1腔体机构开腔体氦检阀/延时关腔体抽气阀（自动单检步）  // 氦检阀开启后腔体压力超过安全阀值，测试判定为NG（氦检异常）
AND H26.06  ; #1-1腔体氦检时腔体压力过高
ORLD
ANDLD
MOVL(498) &1024 D1070  ; #1腔体机构单检步序号  // #1-1腔体出现腔体泄漏，电池泄漏，注氦超时的情况，均跳转至单检步序D1070.10
LD TR0
LD D1070.13  ; #1腔体机构腔体抽气阀打开/延时开#1-2电池抽气阀（自动单检步）
AND T1901  ; #1-1腔体抽真空时间上限到达延时（测试）
AND H26.05  ; #1-2腔体抽真空NG
LD D1070.14  ; #1腔体机构关#1-2电池抽气阀（自动单检步）
AND 822.15  ; #1-2电池抽真空阀关到位标志
LD H26.01  ; #1-2电池泄漏
OR H26.05  ; #1-2腔体抽真空NG
ANDLD
ORLD
LD D1071.00  ; #1腔体机构关#1-2电池注氦阀（自动单检步）
AND 823.01  ; #1-1电池注氦阀关到位标志
AND 823.03  ; #1-2电池注氦阀关到位标志
AND H26.03  ; #1-2电池注氦超时
ORLD
LD D1071.02  ; #1腔体机构开腔体氦检阀/延时关腔体抽气阀（自动单检步）  // 氦检阀开启后腔体压力超过安全阀值，测试判定为NG（氦检异常）
AND H26.07  ; #1-2腔体氦检时腔体压力过高
ORLD
ANDLD
MOVL(498) &524288 D1070  ; #1腔体机构单检步序号  // #1-2腔体出现腔体泄漏，电池泄漏，注氦超时的情况，均跳转至单检步序D1071.03
LD TR0
AND D1071.04  ; #1腔体机构开腔体#1-1阀（自动单检步）
AND 821.00  ; #1-1腔体阀开到位标志
AND 821.02  ; #1-2腔体阀开到位标志
AND 801.11  ; #1腔体氦检阀关到位标志[0001.11]
AND H5.15  ; 腔体模式（0-正压 1-负压）
MOVL(498) &4194304 D1070  ; #1腔体机构单检步序号  // 负压模式下步序正常流程步序不需要抽残气，直接跳转至D1071.06
LD TR0
AND D1070.03  ; #1腔体机构关闭#1-2腔体阀（自动单检步）
ANDNOT H25.00  ; #1-1腔体有料记忆
MOVL(498) &2048 D1070  ; #1腔体机构单检步序号  // 清尾料是#1-1无料，跳转至D1070.11
LD TR0
AND D1070.12  ; #1腔体机构打开#1-2腔体阀（自动单检步）
ANDNOT H25.01  ; #1-2腔体有料记忆
MOVL(498) &1048576 D1070  ; #1腔体机构单检步序号  // 清尾料时#1-2无料，跳转至D1071.04
; rung 19: ******************************* / 清氦步序 / *******************************

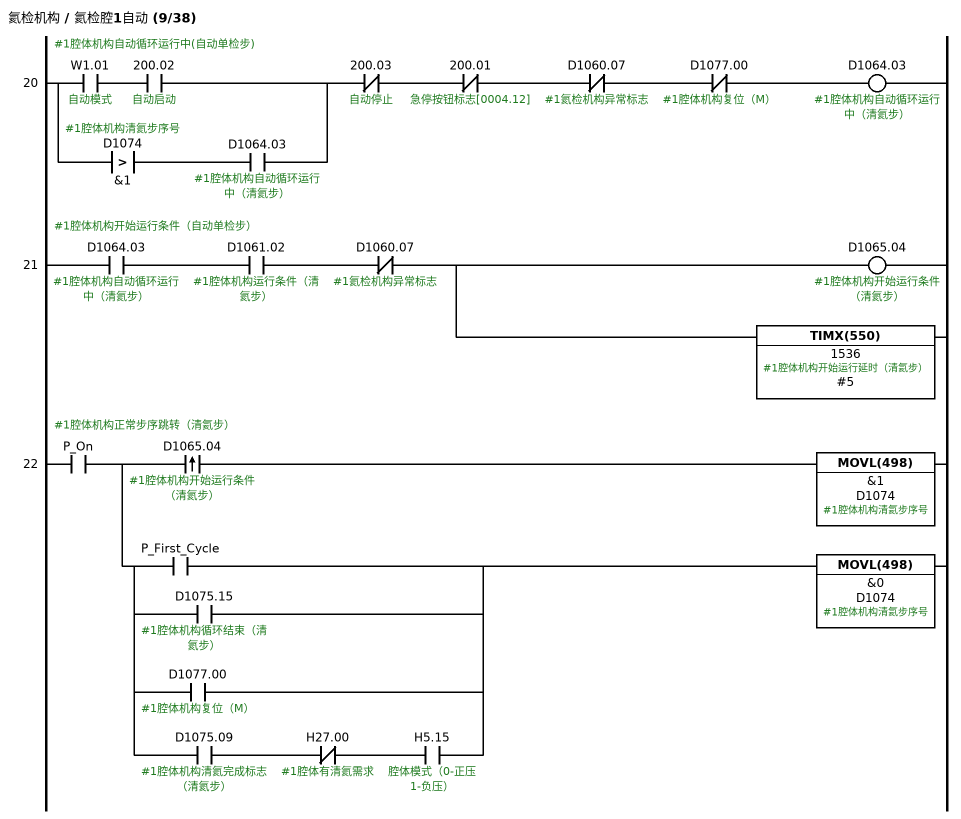
; rung 20: #1腔体机构自动循环运行中(自动单检步)
LD W1.01  ; 自动模式
AND 200.02  ; 自动启动
LD>L(321) D1074 &1  ; #1腔体机构清氦步序号
AND D1064.03  ; #1腔体机构自动循环运行中（清氦步）
ORLD
ANDNOT 200.03  ; 自动停止
ANDNOT 200.01  ; 急停按钮标志[0004.12]
ANDNOT D1060.07  ; #1氦检机构异常标志
ANDNOT D1077.00  ; #1腔体机构复位（M）
OUT D1064.03  ; #1腔体机构自动循环运行中（清氦步）
; rung 21: #1腔体机构开始运行条件（自动单检步）
LD D1064.03  ; #1腔体机构自动循环运行中（清氦步）
AND D1061.02  ; #1腔体机构运行条件（清氦步）
ANDNOT D1060.07  ; #1氦检机构异常标志
OUT D1065.04  ; #1腔体机构开始运行条件（清氦步）
TIMX(550) 1536 #5  ; #1腔体机构开始运行延时（清氦步）
; rung 22: #1腔体机构正常步序跳转（清氦步）
LD P_On
OUT TR0
@AND D1065.04  ; #1腔体机构开始运行条件（清氦步）
MOVL(498) &1 D1074  ; #1腔体机构清氦步序号
LD TR0
LD P_First_Cycle
OR D1075.15  ; #1腔体机构循环结束（清氦步）
OR D1077.00  ; #1腔体机构复位（M）
LD D1075.09  ; #1腔体机构清氦完成标志（清氦步）  // 正压腔体是待料清氦，需跳转回测试步序
ANDNOT H27.00  ; #1腔体有清氦需求
AND H5.15  ; 腔体模式（0-正压 1-负压）
ORLD
ANDLD
MOVL(498) &0 D1074  ; #1腔体机构清氦步序号

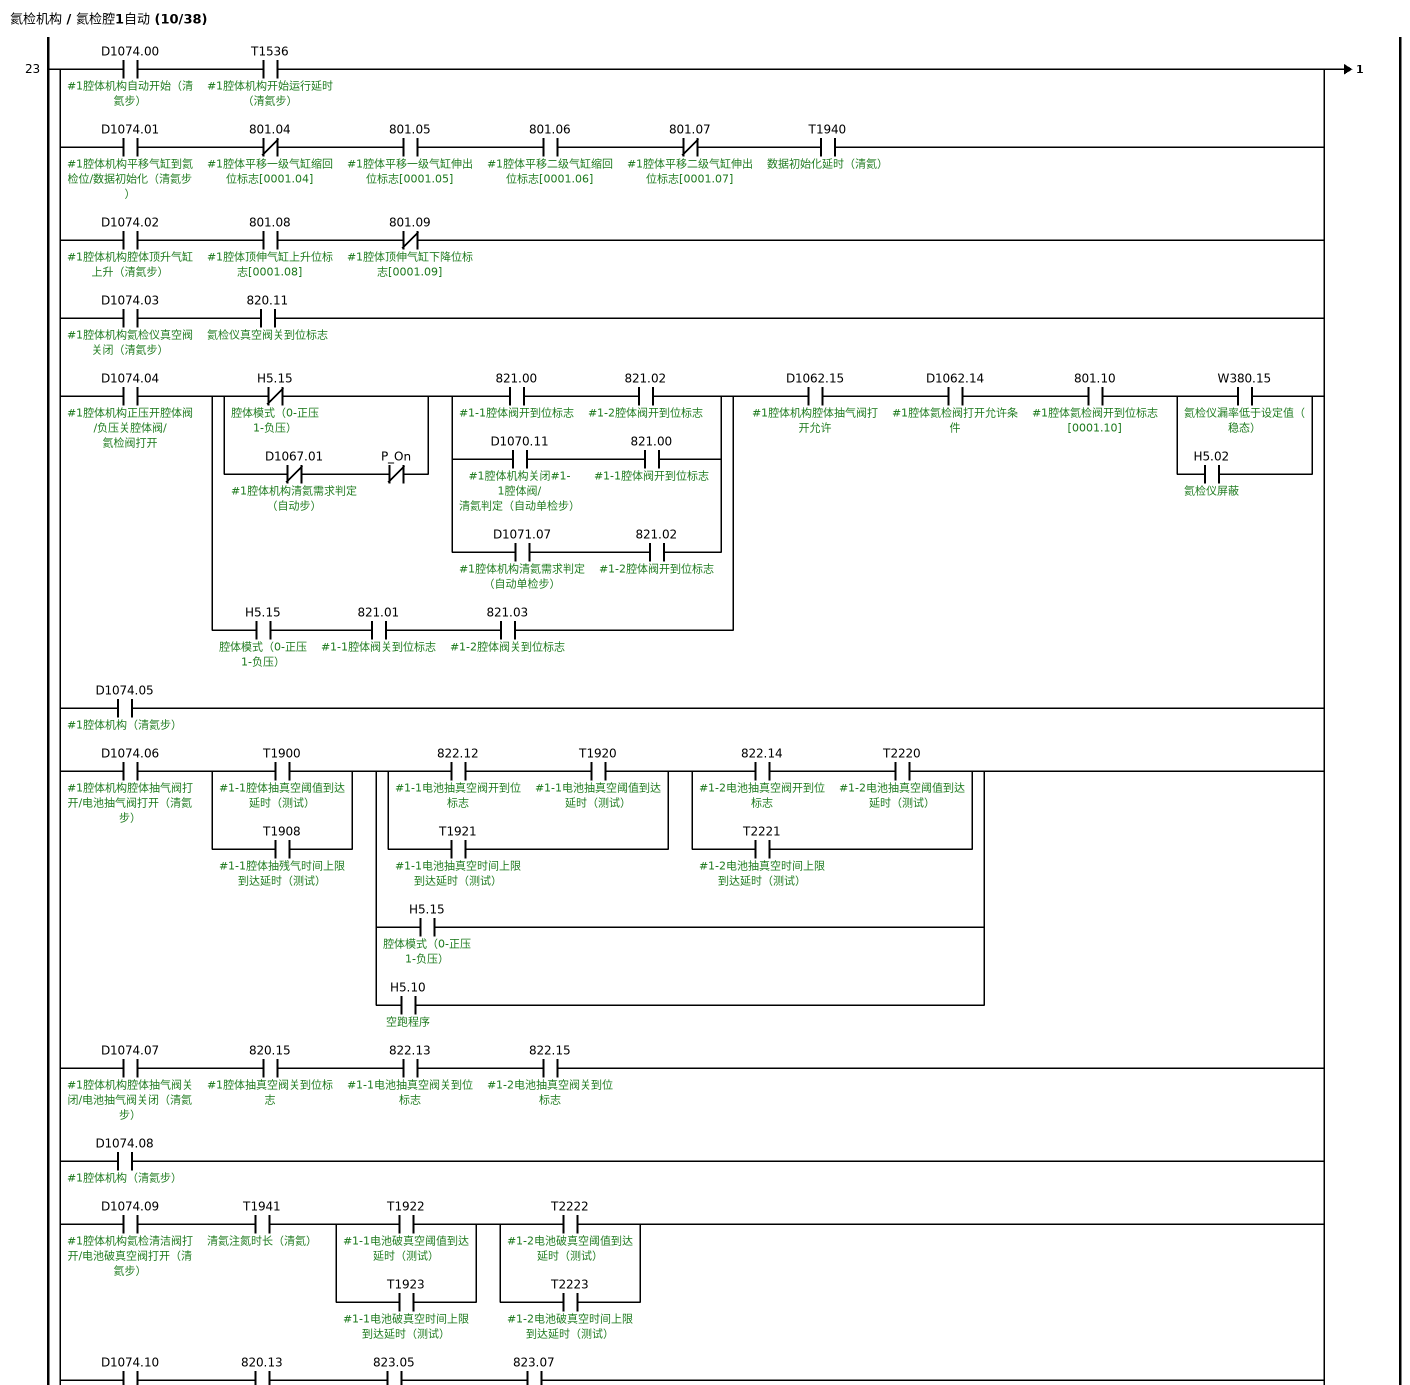

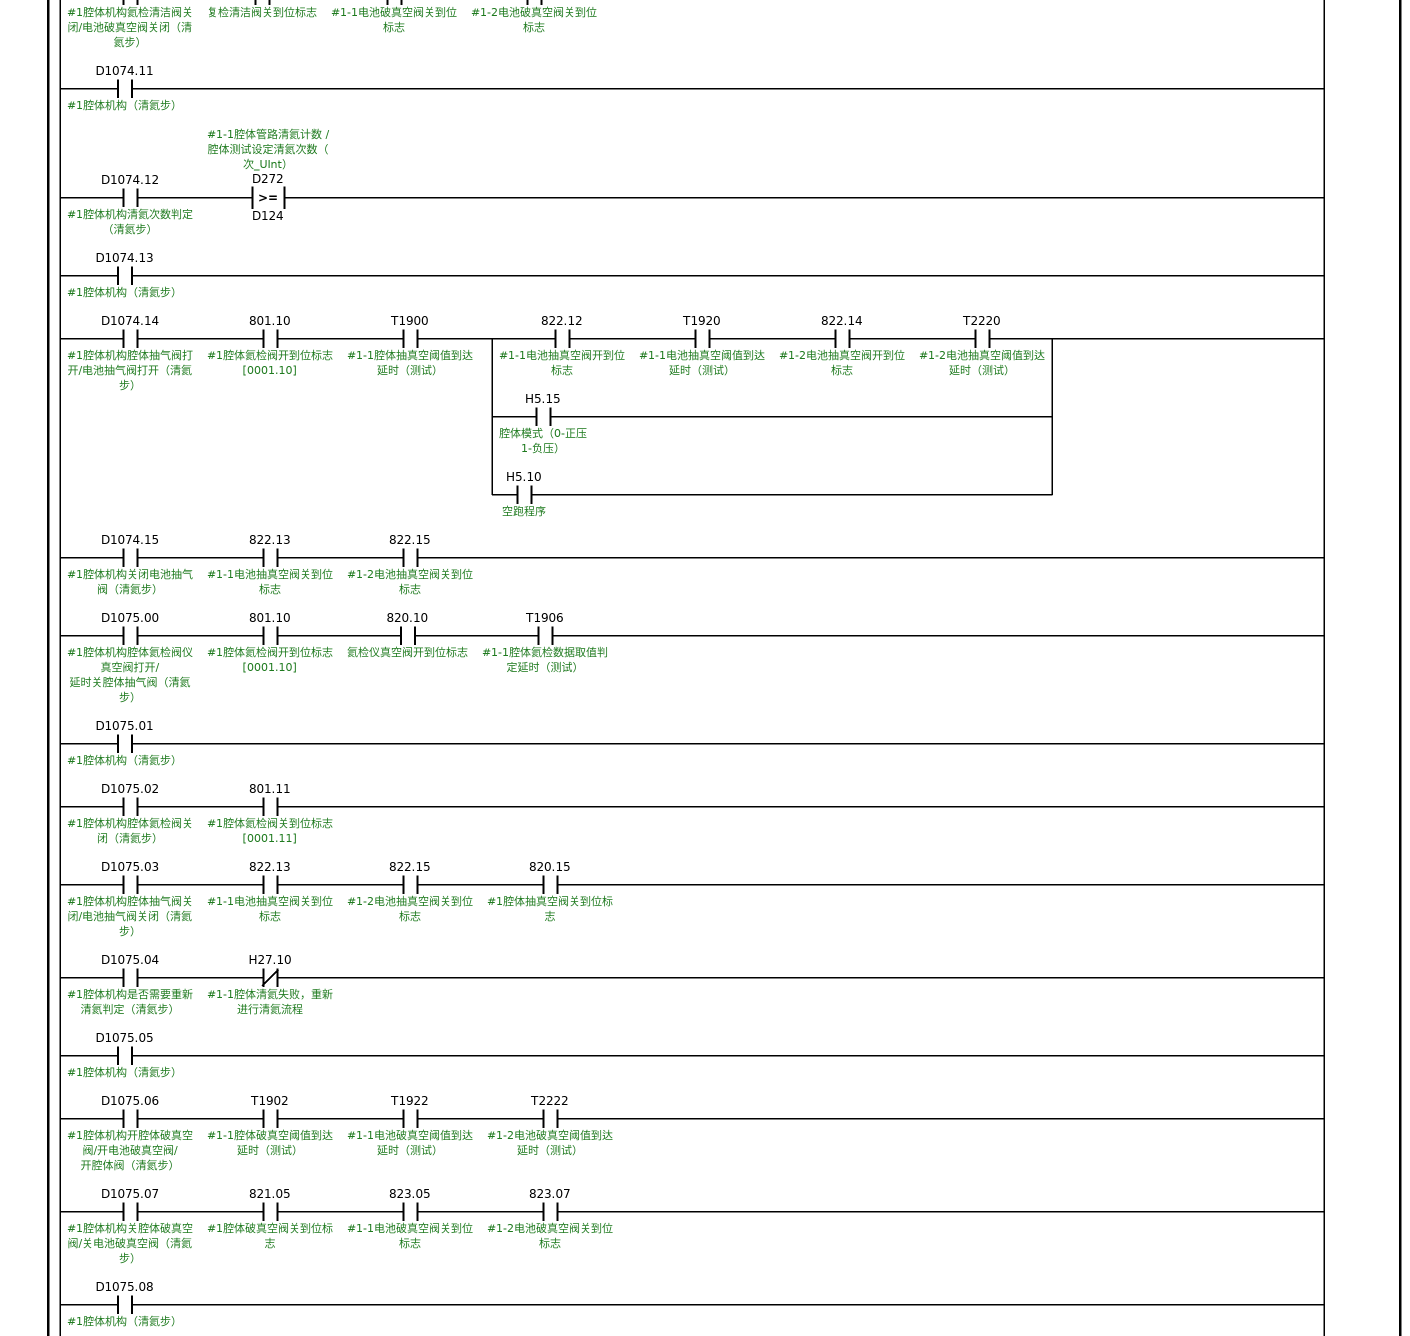

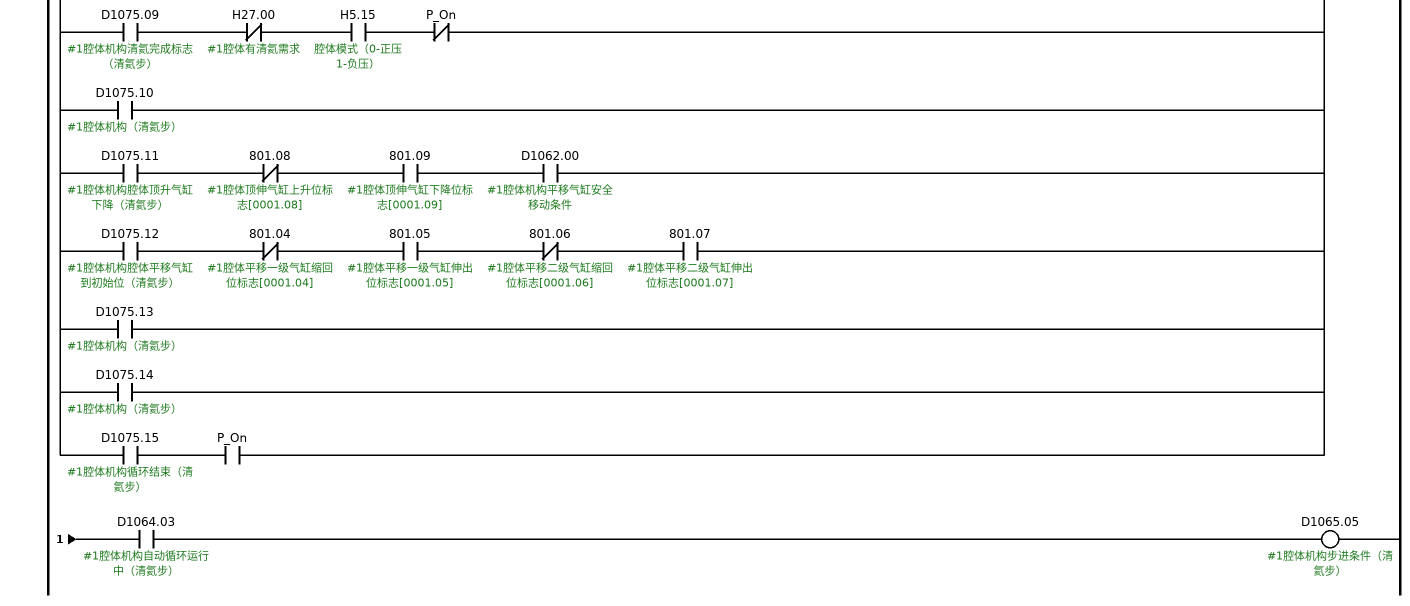
; rung 23
LD D1074.00  ; #1腔体机构自动开始（清氦步）
AND T1536  ; #1腔体机构开始运行延时（清氦步）
LD D1074.01  ; #1腔体机构平移气缸到氦检位/数据初始化（清氦步）
ANDNOT 801.04  ; #1腔体平移一级气缸缩回位标志[0001.04]
AND 801.05  ; #1腔体平移一级气缸伸出位标志[0001.05]
AND 801.06  ; #1腔体平移二级气缸缩回位标志[0001.06]
ANDNOT 801.07  ; #1腔体平移二级气缸伸出位标志[0001.07]
AND T1940  ; 数据初始化延时（清氦）
ORLD
LD D1074.02  ; #1腔体机构腔体顶升气缸上升（清氦步）
AND 801.08  ; #1腔体顶伸气缸上升位标志[0001.08]
ANDNOT 801.09  ; #1腔体顶伸气缸下降位标志[0001.09]
ORLD
LD D1074.03  ; #1腔体机构氦检仪真空阀关闭（清氦步）
AND 820.11  ; 氦检仪真空阀关到位标志
ORLD
LD D1074.04  ; #1腔体机构正压开腔体阀/负压关腔体阀/氦检阀打开  // 负压模式下，复测前的清氦不允许抽电池
LDNOT H5.15  ; 腔体模式（0-正压 1-负压）
LDNOT D1067.01  ; #1腔体机构清氦需求判定（自动步）
ANDNOT P_On
ORLD
LD 821.00  ; #1-1腔体阀开到位标志
AND 821.02  ; #1-2腔体阀开到位标志
LD D1070.11  ; #1腔体机构关闭#1-1腔体阀/清氦判定（自动单检步）
AND 821.00  ; #1-1腔体阀开到位标志
ORLD
LD D1071.07  ; #1腔体机构清氦需求判定（自动单检步）
AND 821.02  ; #1-2腔体阀开到位标志
ORLD
ANDLD
LD H5.15  ; 腔体模式（0-正压 1-负压）
AND 821.01  ; #1-1腔体阀关到位标志
AND 821.03  ; #1-2腔体阀关到位标志
ORLD
ANDLD
AND D1062.15  ; #1腔体机构腔体抽气阀打开允许
AND D1062.14  ; #1腔体氦检阀打开允许条件
AND 801.10  ; #1腔体氦检阀开到位标志[0001.10]
LD W380.15  ; 氦检仪漏率低于设定值（稳态）
OR H5.02  ; 氦检仪屏蔽
ANDLD
ORLD
OR D1074.05  ; #1腔体机构（清氦步）
LD D1074.06  ; #1腔体机构腔体抽气阀打开/电池抽气阀打开（清氦步）
LD T1900  ; #1-1腔体抽真空阈值到达延时（测试）
OR T1908  ; #1-1腔体抽残气时间上限到达延时（测试）
ANDLD
LD 822.12  ; #1-1电池抽真空阀开到位标志
AND T1920  ; #1-1电池抽真空阈值到达延时（测试）
OR T1921  ; #1-1电池抽真空时间上限到达延时（测试）
LD 822.14  ; #1-2电池抽真空阀开到位标志
AND T2220  ; #1-2电池抽真空阈值到达延时（测试）
OR T2221  ; #1-2电池抽真空时间上限到达延时（测试）
ANDLD
OR H5.15  ; 腔体模式（0-正压 1-负压）
OR H5.10  ; 空跑程序
ANDLD
ORLD
LD D1074.07  ; #1腔体机构腔体抽气阀关闭/电池抽气阀关闭（清氦步）
AND 820.15  ; #1腔体抽真空阀关到位标志
AND 822.13  ; #1-1电池抽真空阀关到位标志
AND 822.15  ; #1-2电池抽真空阀关到位标志
ORLD
OR D1074.08  ; #1腔体机构（清氦步）
LD D1074.09  ; #1腔体机构氦检清洁阀打开/电池破真空阀打开（清氦步）
AND T1941  ; 清氦注氮时长（清氦）
LD T1922  ; #1-1电池破真空阈值到达延时（测试）
OR T1923  ; #1-1电池破真空时间上限到达延时（测试）
ANDLD
LD T2222  ; #1-2电池破真空阈值到达延时（测试）
OR T2223  ; #1-2电池破真空时间上限到达延时（测试）
ANDLD
ORLD
LD D1074.10  ; #1腔体机构氦检清洁阀关闭/电池破真空阀关闭（清氦步）
AND 820.13  ; 复检清洁阀关到位标志
AND 823.05  ; #1-1电池破真空阀关到位标志
AND 823.07  ; #1-2电池破真空阀关到位标志
ORLD
OR D1074.11  ; #1腔体机构（清氦步）
LD D1074.12  ; #1腔体机构清氦次数判定（清氦步）
AND>=(325) D272 D124  ; #1-1腔体管路清氦计数, 腔体测试设定清氦次数（次_UInt）
ORLD
OR D1074.13  ; #1腔体机构（清氦步）
LD D1074.14  ; #1腔体机构腔体抽气阀打开/电池抽气阀打开（清氦步）
AND 801.10  ; #1腔体氦检阀开到位标志[0001.10]
AND T1900  ; #1-1腔体抽真空阈值到达延时（测试）
LD 822.12  ; #1-1电池抽真空阀开到位标志
AND T1920  ; #1-1电池抽真空阈值到达延时（测试）
AND 822.14  ; #1-2电池抽真空阀开到位标志
AND T2220  ; #1-2电池抽真空阈值到达延时（测试）
OR H5.15  ; 腔体模式（0-正压 1-负压）
OR H5.10  ; 空跑程序
ANDLD
ORLD
LD D1074.15  ; #1腔体机构关闭电池抽气阀（清氦步）
AND 822.13  ; #1-1电池抽真空阀关到位标志
AND 822.15  ; #1-2电池抽真空阀关到位标志
ORLD
LD D1075.00  ; #1腔体机构腔体氦检阀仪真空阀打开/延时关腔体抽气阀（清氦步）
AND 801.10  ; #1腔体氦检阀开到位标志[0001.10]
AND 820.10  ; 氦检仪真空阀开到位标志
AND T1906  ; #1-1腔体氦检数据取值判定延时（测试）
ORLD
OR D1075.01  ; #1腔体机构（清氦步）
LD D1075.02  ; #1腔体机构腔体氦检阀关闭（清氦步）
AND 801.11  ; #1腔体氦检阀关到位标志[0001.11]
ORLD
LD D1075.03  ; #1腔体机构腔体抽气阀关闭/电池抽气阀关闭（清氦步）
AND 822.13  ; #1-1电池抽真空阀关到位标志
AND 822.15  ; #1-2电池抽真空阀关到位标志
AND 820.15  ; #1腔体抽真空阀关到位标志
ORLD
LD D1075.04  ; #1腔体机构是否需要重新清氦判定（清氦步）
ANDNOT H27.10  ; #1-1腔体清氦失败，重新进行清氦流程  // 清氦失败，重新进行清氦
ORLD
OR D1075.05  ; #1腔体机构（清氦步）
LD D1075.06  ; #1腔体机构开腔体破真空阀/开电池破真空阀/开腔体阀（清氦步）
AND T1902  ; #1-1腔体破真空阈值到达延时（测试）
AND T1922  ; #1-1电池破真空阈值到达延时（测试）
AND T2222  ; #1-2电池破真空阈值到达延时（测试）
ORLD
LD D1075.07  ; #1腔体机构关腔体破真空阀/关电池破真空阀（清氦步）
AND 821.05  ; #1腔体破真空阀关到位标志
AND 823.05  ; #1-1电池破真空阀关到位标志
AND 823.07  ; #1-2电池破真空阀关到位标志
ORLD
OR D1075.08  ; #1腔体机构（清氦步）
LD D1075.09  ; #1腔体机构清氦完成标志（清氦步）  // 正压腔体是待料清氦，需跳转回测试步序
ANDNOT H27.00  ; #1腔体有清氦需求
AND H5.15  ; 腔体模式（0-正压 1-负压）
ANDNOT P_On
ORLD
OR D1075.10  ; #1腔体机构（清氦步）
LD D1075.11  ; #1腔体机构腔体顶升气缸下降（清氦步）
ANDNOT 801.08  ; #1腔体顶伸气缸上升位标志[0001.08]
AND 801.09  ; #1腔体顶伸气缸下降位标志[0001.09]
AND D1062.00  ; #1腔体机构平移气缸安全移动条件
ORLD
LD D1075.12  ; #1腔体机构腔体平移气缸到初始位（清氦步）
ANDNOT 801.04  ; #1腔体平移一级气缸缩回位标志[0001.04]
AND 801.05  ; #1腔体平移一级气缸伸出位标志[0001.05]
ANDNOT 801.06  ; #1腔体平移二级气缸缩回位标志[0001.06]
AND 801.07  ; #1腔体平移二级气缸伸出位标志[0001.07]
ORLD
OR D1075.13  ; #1腔体机构（清氦步）
OR D1075.14  ; #1腔体机构（清氦步）
LD D1075.15  ; #1腔体机构循环结束（清氦步）
AND P_On
ORLD
AND D1064.03  ; #1腔体机构自动循环运行中（清氦步）
OUT D1065.05  ; #1腔体机构步进条件（清氦步）

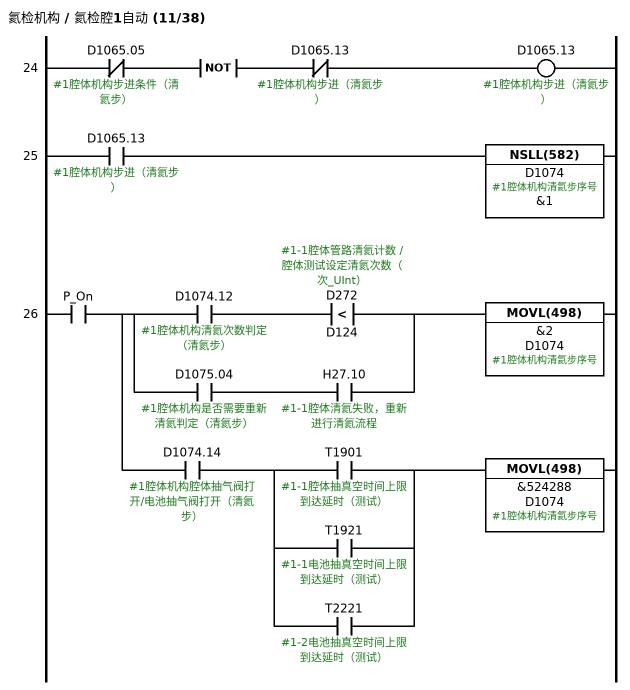
; rung 24
LDNOT D1065.05  ; #1腔体机构步进条件（清氦步）
NOT(520)
ANDNOT D1065.13  ; #1腔体机构步进（清氦步）
OUT D1065.13  ; #1腔体机构步进（清氦步）
; rung 25
LD D1065.13  ; #1腔体机构步进（清氦步）
NSLL(582) D1074 &1  ; #1腔体机构清氦步序号
; rung 26
LD P_On
OUT TR0
LD D1074.12  ; #1腔体机构清氦次数判定（清氦步）
AND<(310) D272 D124  ; #1-1腔体管路清氦计数, 腔体测试设定清氦次数（次_UInt）
LD D1075.04  ; #1腔体机构是否需要重新清氦判定（清氦步）
AND H27.10  ; #1-1腔体清氦失败，重新进行清氦流程  // 清氦失败，重新进行清氦
ORLD
ANDLD
MOVL(498) &2 D1074  ; #1腔体机构清氦步序号
LD TR0
AND D1074.14  ; #1腔体机构腔体抽气阀打开/电池抽气阀打开（清氦步）
LD T1901  ; #1-1腔体抽真空时间上限到达延时（测试）
OR T1921  ; #1-1电池抽真空时间上限到达延时（测试）
OR T2221  ; #1-2电池抽真空时间上限到达延时（测试）
ANDLD
MOVL(498) &524288 D1074  ; #1腔体机构清氦步序号  // 清氦过程腔体或电池抽气上限达到，均直接判定清氦完成，不进入氦检步序（跳转至D1075.03）

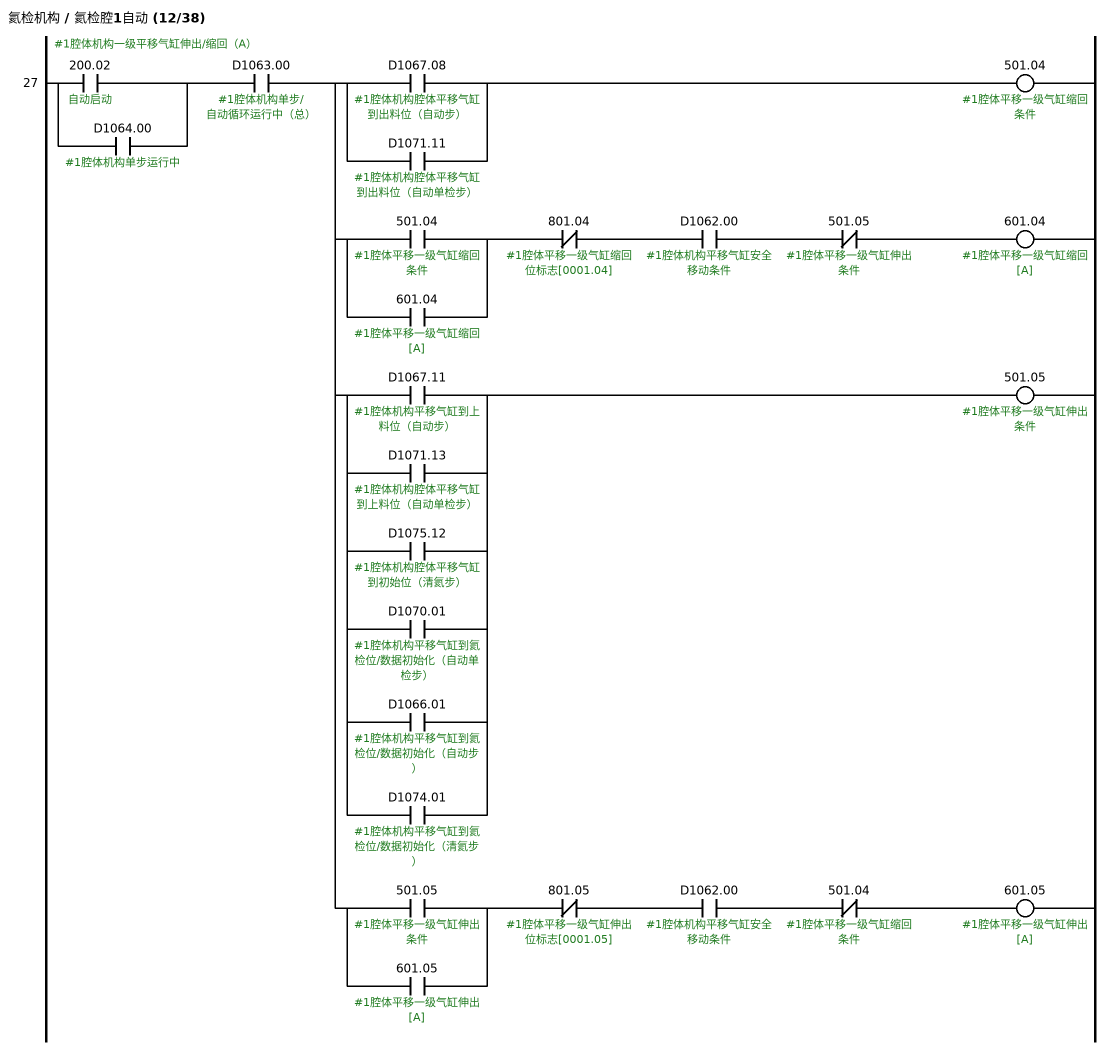
; rung 27: #1腔体机构一级平移气缸伸出/缩回（A）
LD 200.02  ; 自动启动
OR D1064.00  ; #1腔体机构单步运行中
AND D1063.00  ; #1腔体机构单步/自动循环运行中（总）
OUT TR0
LD D1067.08  ; #1腔体机构腔体平移气缸到出料位（自动步）
OR D1071.11  ; #1腔体机构腔体平移气缸到出料位（自动单检步）
ANDLD
OUT 501.04  ; #1腔体平移一级气缸缩回条件
LD TR0
LD 501.04  ; #1腔体平移一级气缸缩回条件
OR 601.04  ; #1腔体平移一级气缸缩回[A]
ANDLD
ANDNOT 801.04  ; #1腔体平移一级气缸缩回位标志[0001.04]
AND D1062.00  ; #1腔体机构平移气缸安全移动条件
ANDNOT 501.05  ; #1腔体平移一级气缸伸出条件
OUT 601.04  ; #1腔体平移一级气缸缩回[A]
LD TR0
LD D1067.11  ; #1腔体机构平移气缸到上料位（自动步）
OR D1071.13  ; #1腔体机构腔体平移气缸到上料位（自动单检步）
OR D1075.12  ; #1腔体机构腔体平移气缸到初始位（清氦步）
OR D1070.01  ; #1腔体机构平移气缸到氦检位/数据初始化（自动单检步）
OR D1066.01  ; #1腔体机构平移气缸到氦检位/数据初始化（自动步）
OR D1074.01  ; #1腔体机构平移气缸到氦检位/数据初始化（清氦步）
ANDLD
OUT 501.05  ; #1腔体平移一级气缸伸出条件
LD TR0
LD 501.05  ; #1腔体平移一级气缸伸出条件
OR 601.05  ; #1腔体平移一级气缸伸出[A]
ANDLD
ANDNOT 801.05  ; #1腔体平移一级气缸伸出位标志[0001.05]
AND D1062.00  ; #1腔体机构平移气缸安全移动条件
ANDNOT 501.04  ; #1腔体平移一级气缸缩回条件
OUT 601.05  ; #1腔体平移一级气缸伸出[A]

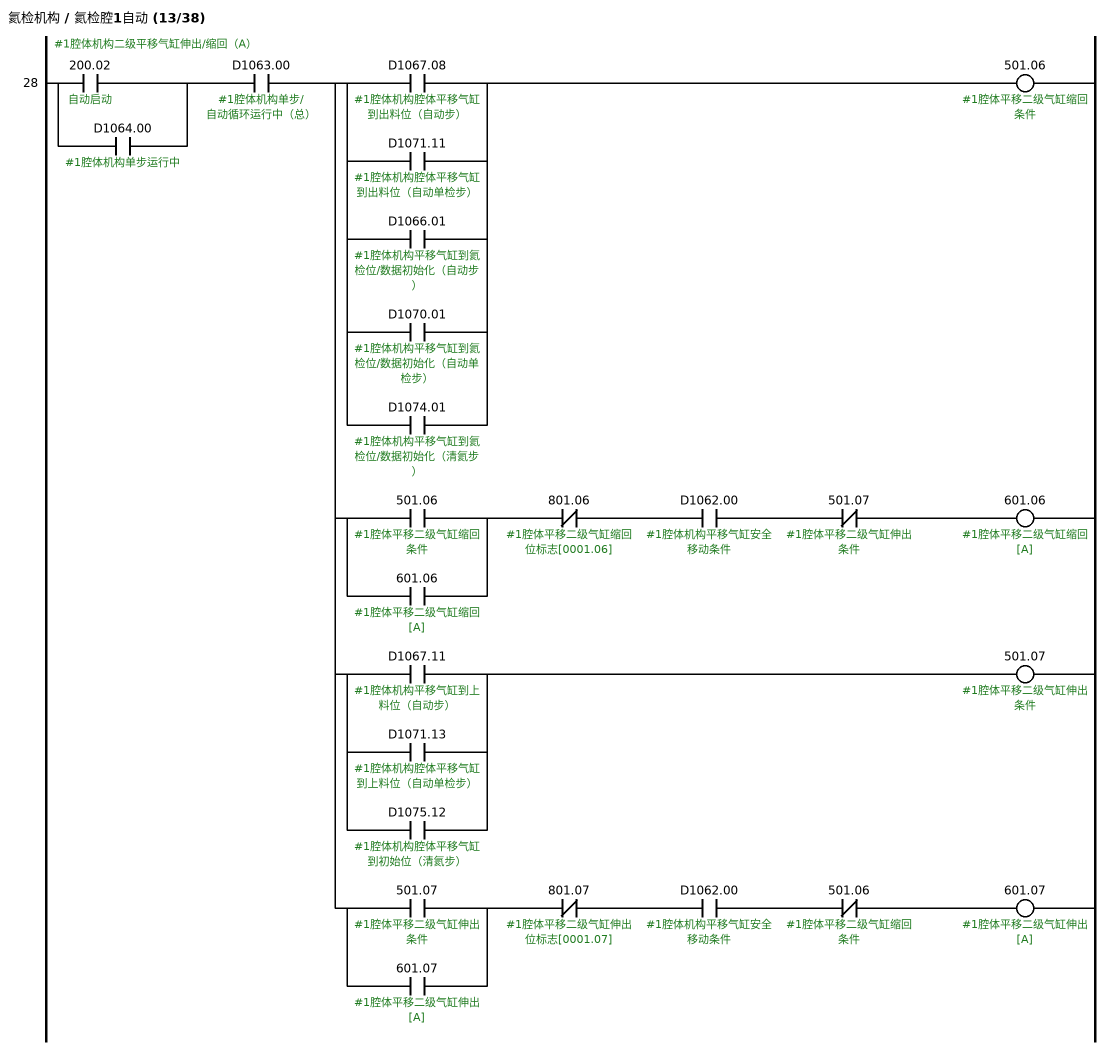
; rung 28: #1腔体机构二级平移气缸伸出/缩回（A）
LD 200.02  ; 自动启动
OR D1064.00  ; #1腔体机构单步运行中
AND D1063.00  ; #1腔体机构单步/自动循环运行中（总）
OUT TR0
LD D1067.08  ; #1腔体机构腔体平移气缸到出料位（自动步）
OR D1071.11  ; #1腔体机构腔体平移气缸到出料位（自动单检步）
OR D1066.01  ; #1腔体机构平移气缸到氦检位/数据初始化（自动步）
OR D1070.01  ; #1腔体机构平移气缸到氦检位/数据初始化（自动单检步）
OR D1074.01  ; #1腔体机构平移气缸到氦检位/数据初始化（清氦步）
ANDLD
OUT 501.06  ; #1腔体平移二级气缸缩回条件
LD TR0
LD 501.06  ; #1腔体平移二级气缸缩回条件
OR 601.06  ; #1腔体平移二级气缸缩回[A]
ANDLD
ANDNOT 801.06  ; #1腔体平移二级气缸缩回位标志[0001.06]
AND D1062.00  ; #1腔体机构平移气缸安全移动条件
ANDNOT 501.07  ; #1腔体平移二级气缸伸出条件
OUT 601.06  ; #1腔体平移二级气缸缩回[A]
LD TR0
LD D1067.11  ; #1腔体机构平移气缸到上料位（自动步）
OR D1071.13  ; #1腔体机构腔体平移气缸到上料位（自动单检步）
OR D1075.12  ; #1腔体机构腔体平移气缸到初始位（清氦步）
ANDLD
OUT 501.07  ; #1腔体平移二级气缸伸出条件
LD TR0
LD 501.07  ; #1腔体平移二级气缸伸出条件
OR 601.07  ; #1腔体平移二级气缸伸出[A]
ANDLD
ANDNOT 801.07  ; #1腔体平移二级气缸伸出位标志[0001.07]
AND D1062.00  ; #1腔体机构平移气缸安全移动条件
ANDNOT 501.06  ; #1腔体平移二级气缸缩回条件
OUT 601.07  ; #1腔体平移二级气缸伸出[A]

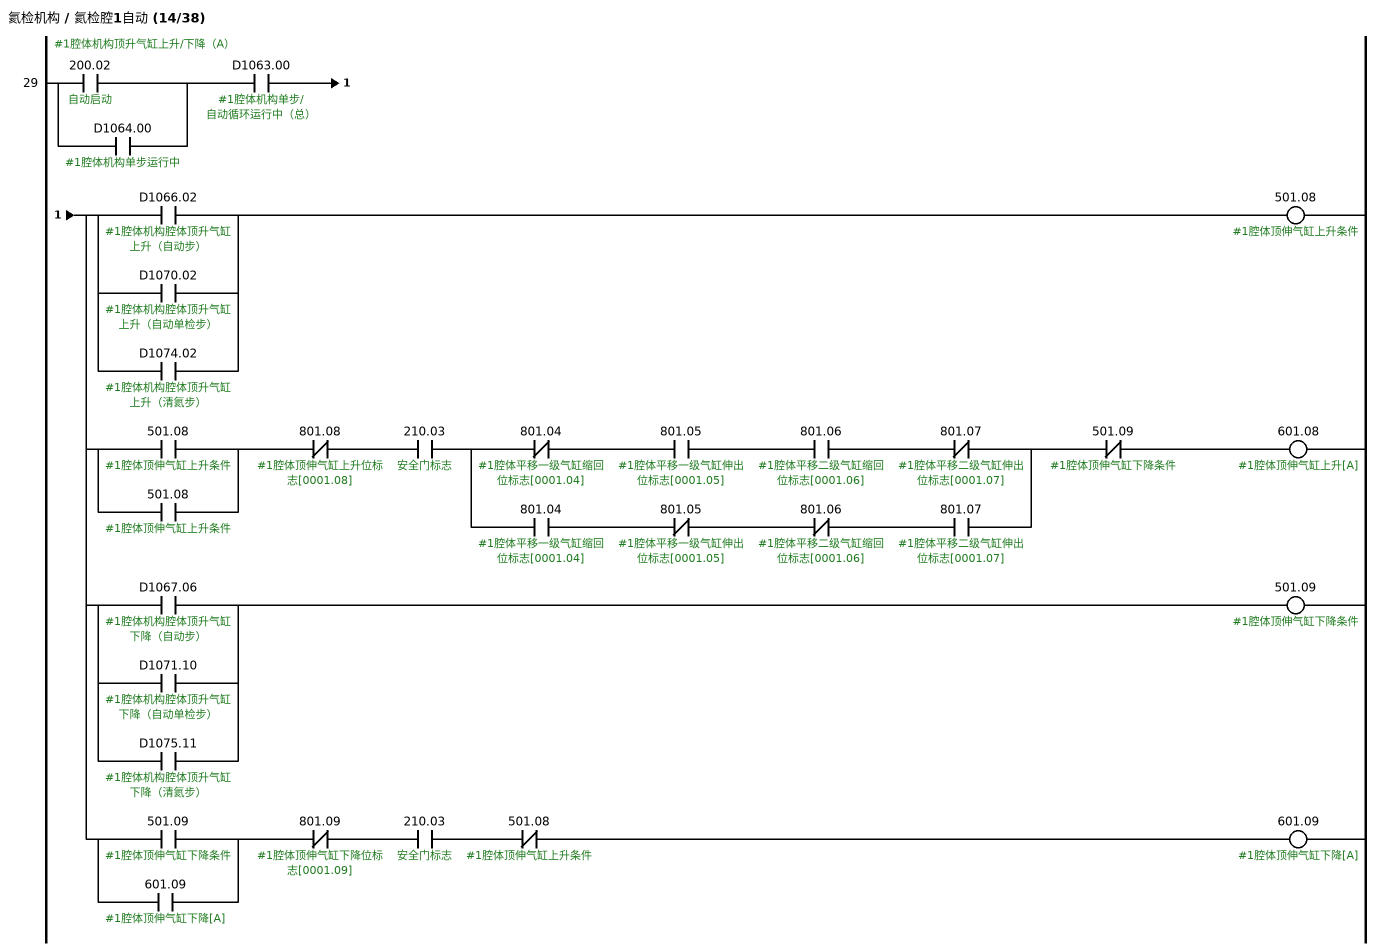
; rung 29: #1腔体机构顶升气缸上升/下降（A）
LD 200.02  ; 自动启动
OR D1064.00  ; #1腔体机构单步运行中
AND D1063.00  ; #1腔体机构单步/自动循环运行中（总）
OUT TR0
LD D1066.02  ; #1腔体机构腔体顶升气缸上升（自动步）
OR D1070.02  ; #1腔体机构腔体顶升气缸上升（自动单检步）
OR D1074.02  ; #1腔体机构腔体顶升气缸上升（清氦步）
ANDLD
OUT 501.08  ; #1腔体顶伸气缸上升条件
LD TR0
LD 501.08  ; #1腔体顶伸气缸上升条件
OR 501.08  ; #1腔体顶伸气缸上升条件
ANDLD
ANDNOT 801.08  ; #1腔体顶伸气缸上升位标志[0001.08]
AND 210.03  ; 安全门标志
LDNOT 801.04  ; #1腔体平移一级气缸缩回位标志[0001.04]
AND 801.05  ; #1腔体平移一级气缸伸出位标志[0001.05]
AND 801.06  ; #1腔体平移二级气缸缩回位标志[0001.06]
ANDNOT 801.07  ; #1腔体平移二级气缸伸出位标志[0001.07]
LD 801.04  ; #1腔体平移一级气缸缩回位标志[0001.04]
ANDNOT 801.05  ; #1腔体平移一级气缸伸出位标志[0001.05]
ANDNOT 801.06  ; #1腔体平移二级气缸缩回位标志[0001.06]
AND 801.07  ; #1腔体平移二级气缸伸出位标志[0001.07]
ORLD
ANDLD
ANDNOT 501.09  ; #1腔体顶伸气缸下降条件
OUT 601.08  ; #1腔体顶伸气缸上升[A]
LD TR0
LD D1067.06  ; #1腔体机构腔体顶升气缸下降（自动步）
OR D1071.10  ; #1腔体机构腔体顶升气缸下降（自动单检步）
OR D1075.11  ; #1腔体机构腔体顶升气缸下降（清氦步）
ANDLD
OUT 501.09  ; #1腔体顶伸气缸下降条件
LD TR0
LD 501.09  ; #1腔体顶伸气缸下降条件
OR 601.09  ; #1腔体顶伸气缸下降[A]
ANDLD
ANDNOT 801.09  ; #1腔体顶伸气缸下降位标志[0001.09]
AND 210.03  ; 安全门标志
ANDNOT 501.08  ; #1腔体顶伸气缸上升条件
OUT 601.09  ; #1腔体顶伸气缸下降[A]

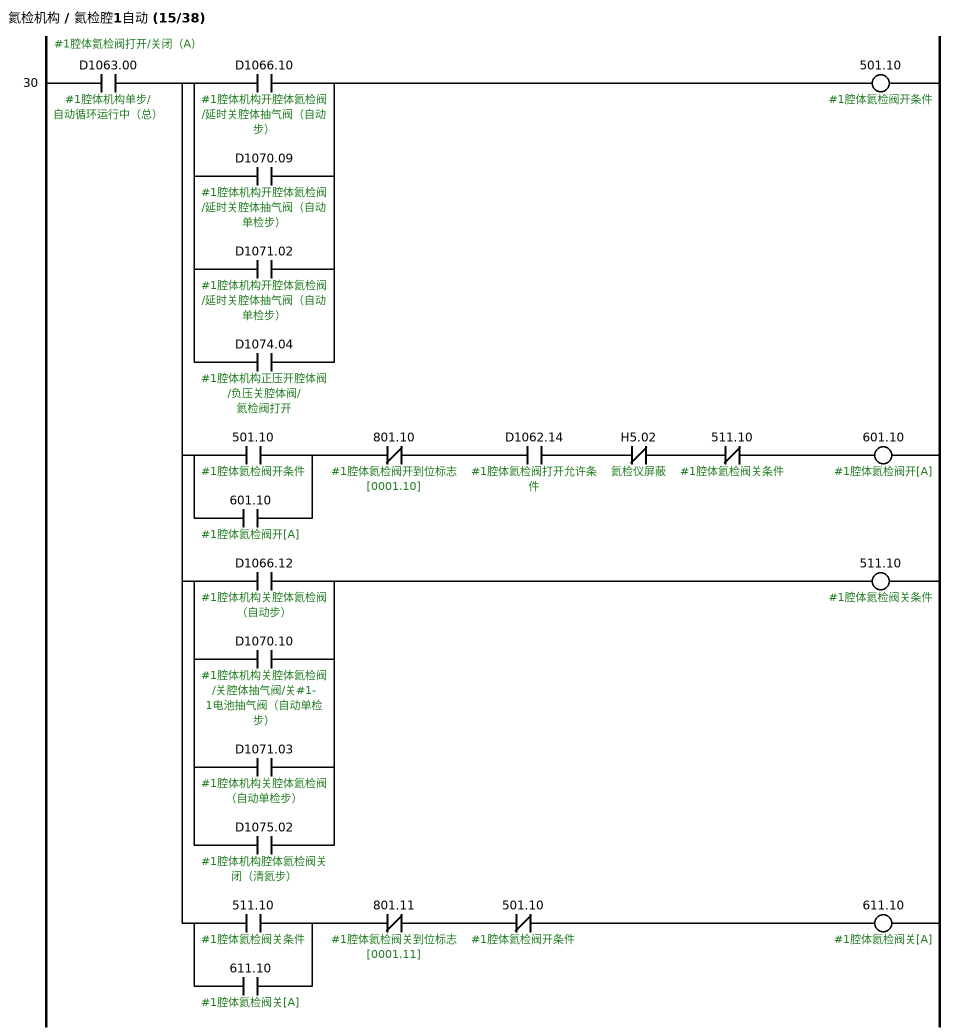
; rung 30: #1腔体氦检阀打开/关闭（A）
LD D1063.00  ; #1腔体机构单步/自动循环运行中（总）
OUT TR0
LD D1066.10  ; #1腔体机构开腔体氦检阀/延时关腔体抽气阀（自动步）
OR D1070.09  ; #1腔体机构开腔体氦检阀/延时关腔体抽气阀（自动单检步）
OR D1071.02  ; #1腔体机构开腔体氦检阀/延时关腔体抽气阀（自动单检步）
OR D1074.04  ; #1腔体机构正压开腔体阀/负压关腔体阀/氦检阀打开
ANDLD
OUT 501.10  ; #1腔体氦检阀开条件
LD TR0
LD 501.10  ; #1腔体氦检阀开条件
OR 601.10  ; #1腔体氦检阀开[A]
ANDLD
ANDNOT 801.10  ; #1腔体氦检阀开到位标志[0001.10]
AND D1062.14  ; #1腔体氦检阀打开允许条件
ANDNOT H5.02  ; 氦检仪屏蔽
ANDNOT 511.10  ; #1腔体氦检阀关条件
OUT 601.10  ; #1腔体氦检阀开[A]
LD TR0
LD D1066.12  ; #1腔体机构关腔体氦检阀（自动步）
OR D1070.10  ; #1腔体机构关腔体氦检阀/关腔体抽气阀/关#1-1电池抽气阀（自动单检步）
OR D1071.03  ; #1腔体机构关腔体氦检阀（自动单检步）
OR D1075.02  ; #1腔体机构腔体氦检阀关闭（清氦步）
ANDLD
OUT 511.10  ; #1腔体氦检阀关条件
LD TR0
LD 511.10  ; #1腔体氦检阀关条件
OR 611.10  ; #1腔体氦检阀关[A]
ANDLD
ANDNOT 801.11  ; #1腔体氦检阀关到位标志[0001.11]
ANDNOT 501.10  ; #1腔体氦检阀开条件
OUT 611.10  ; #1腔体氦检阀关[A]

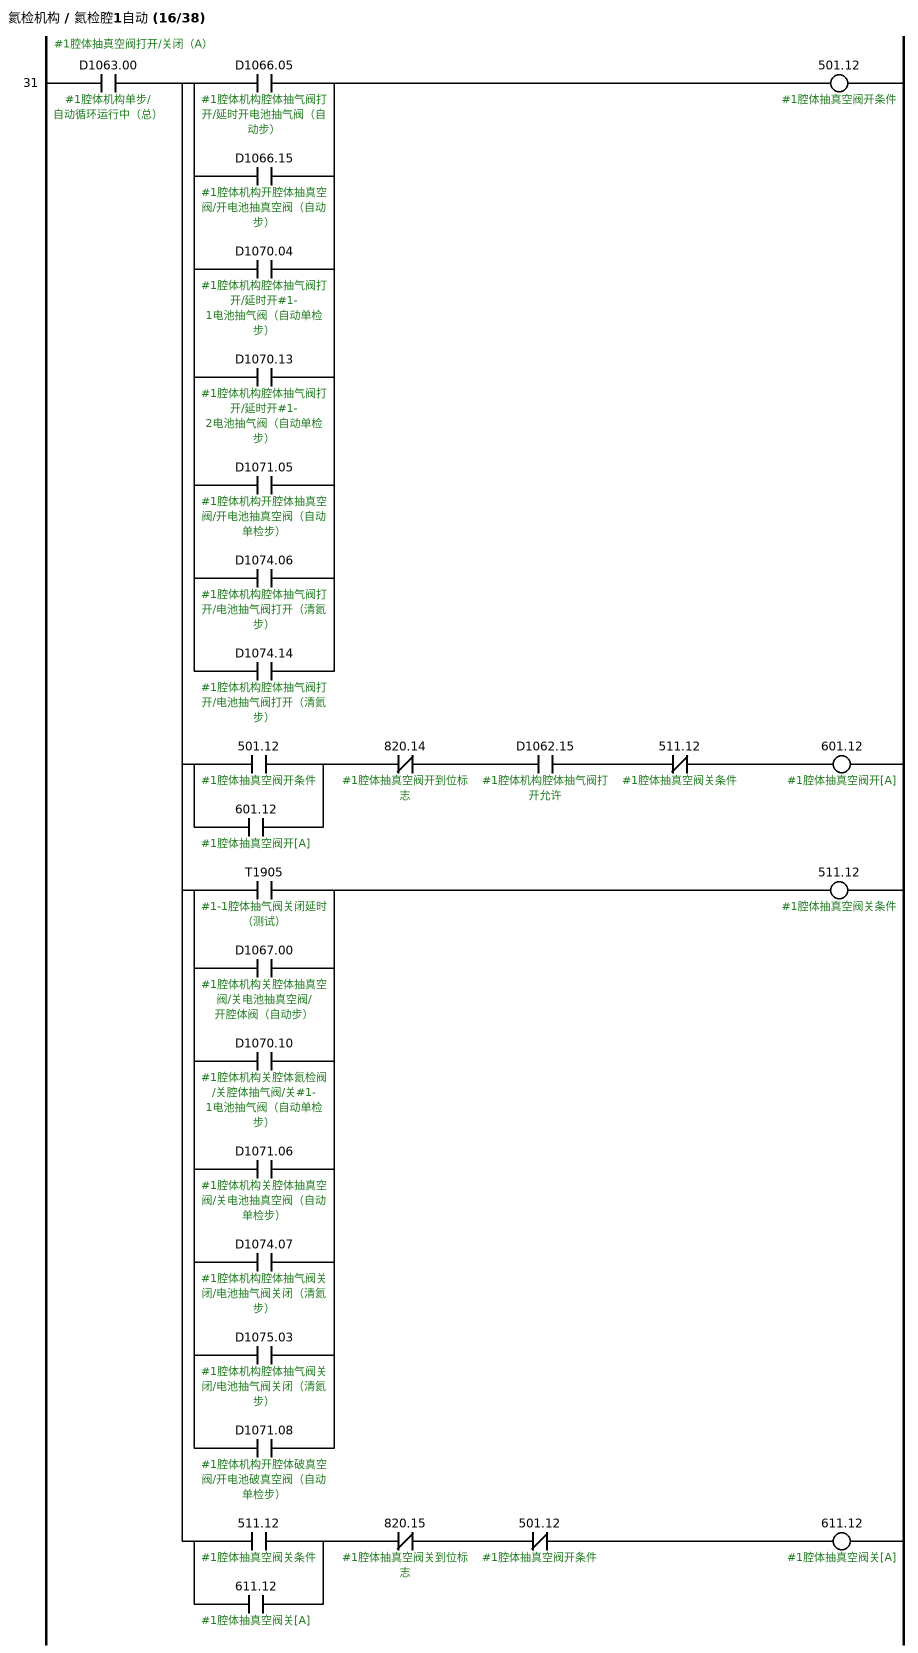
; rung 31: #1腔体抽真空阀打开/关闭（A）
LD D1063.00  ; #1腔体机构单步/自动循环运行中（总）
OUT TR0
LD D1066.05  ; #1腔体机构腔体抽气阀打开/延时开电池抽气阀（自动步）
OR D1066.15  ; #1腔体机构开腔体抽真空阀/开电池抽真空阀（自动步）
OR D1070.04  ; #1腔体机构腔体抽气阀打开/延时开#1-1电池抽气阀（自动单检步）
OR D1070.13  ; #1腔体机构腔体抽气阀打开/延时开#1-2电池抽气阀（自动单检步）
OR D1071.05  ; #1腔体机构开腔体抽真空阀/开电池抽真空阀（自动单检步）
OR D1074.06  ; #1腔体机构腔体抽气阀打开/电池抽气阀打开（清氦步）
OR D1074.14  ; #1腔体机构腔体抽气阀打开/电池抽气阀打开（清氦步）
ANDLD
OUT 501.12  ; #1腔体抽真空阀开条件
LD TR0
LD 501.12  ; #1腔体抽真空阀开条件
OR 601.12  ; #1腔体抽真空阀开[A]
ANDLD
ANDNOT 820.14  ; #1腔体抽真空阀开到位标志
AND D1062.15  ; #1腔体机构腔体抽气阀打开允许
ANDNOT 511.12  ; #1腔体抽真空阀关条件
OUT 601.12  ; #1腔体抽真空阀开[A]
LD TR0
LD T1905  ; #1-1腔体抽气阀关闭延时（测试）
OR D1067.00  ; #1腔体机构关腔体抽真空阀/关电池抽真空阀/开腔体阀（自动步）
OR D1070.10  ; #1腔体机构关腔体氦检阀/关腔体抽气阀/关#1-1电池抽气阀（自动单检步）
OR D1071.06  ; #1腔体机构关腔体抽真空阀/关电池抽真空阀（自动单检步）
OR D1074.07  ; #1腔体机构腔体抽气阀关闭/电池抽气阀关闭（清氦步）
OR D1075.03  ; #1腔体机构腔体抽气阀关闭/电池抽气阀关闭（清氦步）
OR D1071.08  ; #1腔体机构开腔体破真空阀/开电池破真空阀（自动单检步）
ANDLD
OUT 511.12  ; #1腔体抽真空阀关条件
LD TR0
LD 511.12  ; #1腔体抽真空阀关条件
OR 611.12  ; #1腔体抽真空阀关[A]
ANDLD
ANDNOT 820.15  ; #1腔体抽真空阀关到位标志
ANDNOT 501.12  ; #1腔体抽真空阀开条件
OUT 611.12  ; #1腔体抽真空阀关[A]

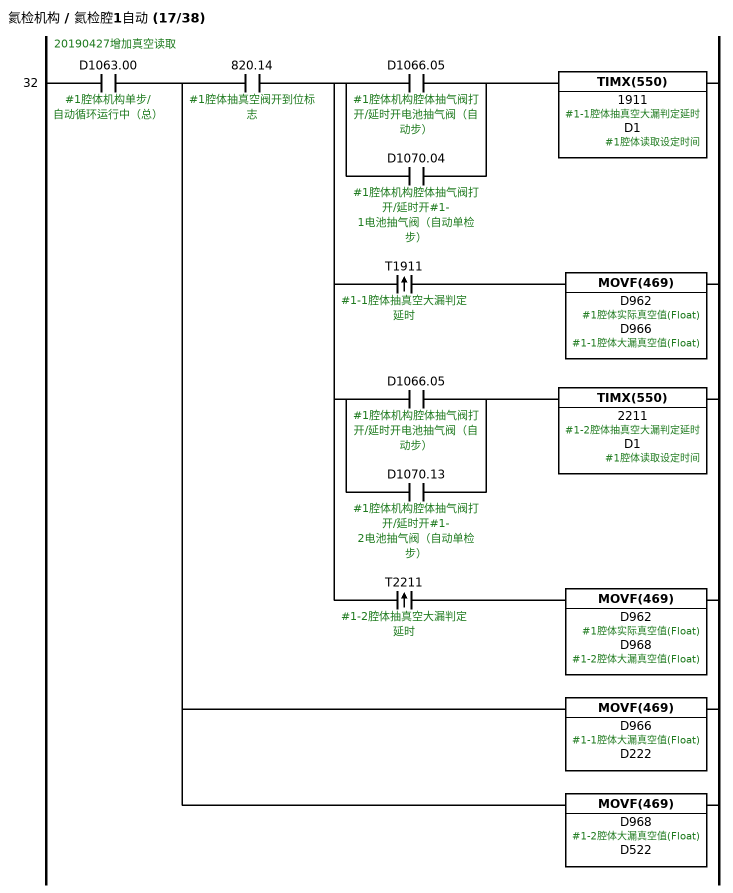
; rung 32: 20190427增加真空读取
LD D1063.00  ; #1腔体机构单步/自动循环运行中（总）
OUT TR0
AND 820.14  ; #1腔体抽真空阀开到位标志
OUT TR1
LD D1066.05  ; #1腔体机构腔体抽气阀打开/延时开电池抽气阀（自动步）
OR D1070.04  ; #1腔体机构腔体抽气阀打开/延时开#1-1电池抽气阀（自动单检步）
ANDLD
TIMX(550) 1911 D1  ; #1腔体读取设定时间, #1-1腔体抽真空大漏判定延时
LD TR1
@AND T1911  ; #1-1腔体抽真空大漏判定延时
MOVF(469) D962 D966  ; #1腔体实际真空值(Float), #1-1腔体大漏真空值(Float)
LD TR1
LD D1066.05  ; #1腔体机构腔体抽气阀打开/延时开电池抽气阀（自动步）
OR D1070.13  ; #1腔体机构腔体抽气阀打开/延时开#1-2电池抽气阀（自动单检步）
ANDLD
TIMX(550) 2211 D1  ; #1腔体读取设定时间, #1-2腔体抽真空大漏判定延时
LD TR1
@AND T2211  ; #1-2腔体抽真空大漏判定延时
MOVF(469) D962 D968  ; #1腔体实际真空值(Float), #1-2腔体大漏真空值(Float)
LD TR0
MOVF(469) D966 D222  ; #1-1腔体大漏真空值(Float)
MOVF(469) D968 D522  ; #1-2腔体大漏真空值(Float)

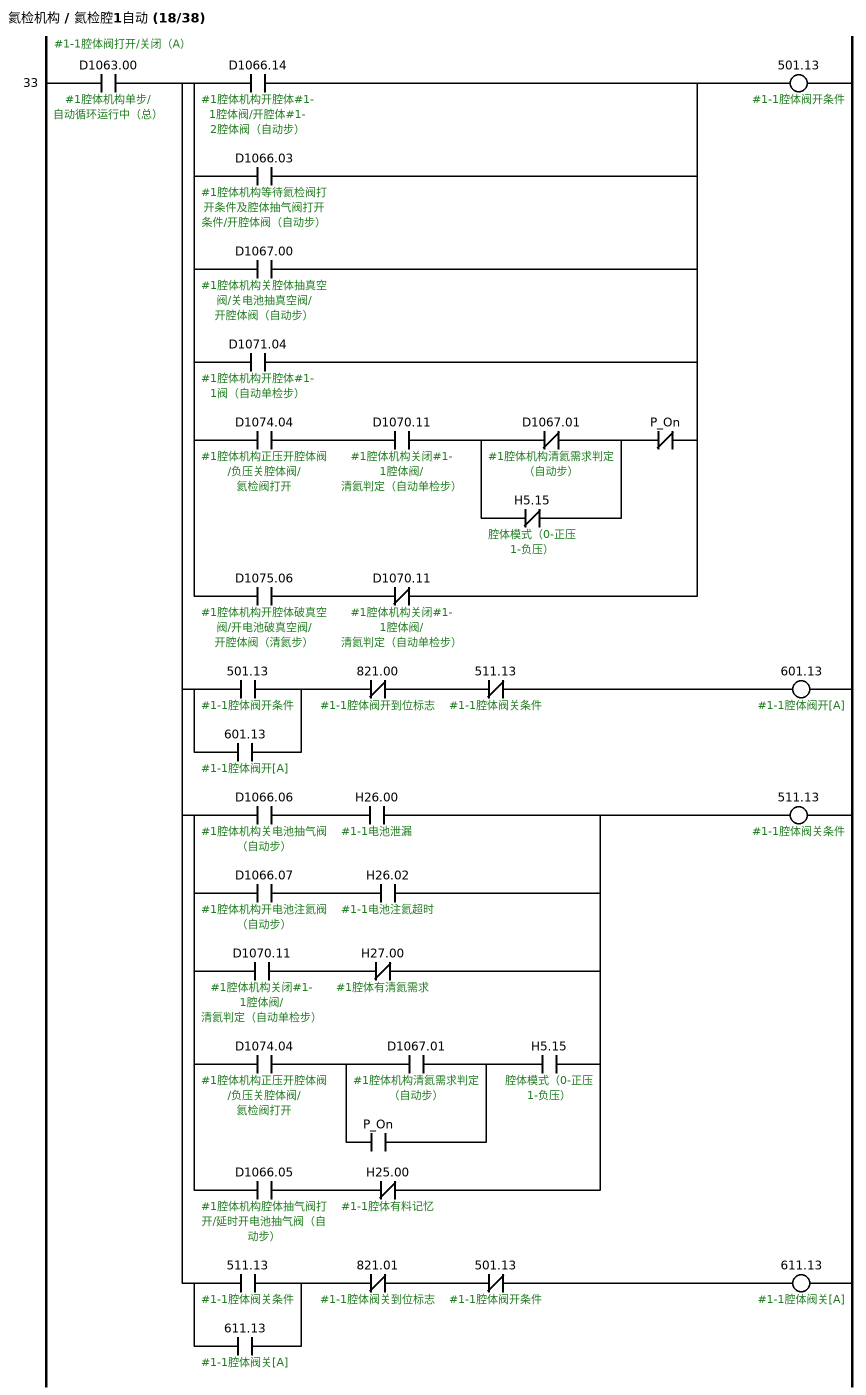
; rung 33: #1-1腔体阀打开/关闭（A）
LD D1063.00  ; #1腔体机构单步/自动循环运行中（总）
OUT TR0
LD D1066.14  ; #1腔体机构开腔体#1-1腔体阀/开腔体#1-2腔体阀（自动步）
OR D1066.03  ; #1腔体机构等待氦检阀打开条件及腔体抽气阀打开条件/开腔体阀（自动步）
OR D1067.00  ; #1腔体机构关腔体抽真空阀/关电池抽真空阀/开腔体阀（自动步）
OR D1071.04  ; #1腔体机构开腔体#1-1阀（自动单检步）
LD D1074.04  ; #1腔体机构正压开腔体阀/负压关腔体阀/氦检阀打开
AND D1070.11  ; #1腔体机构关闭#1-1腔体阀/清氦判定（自动单检步）
LDNOT D1067.01  ; #1腔体机构清氦需求判定（自动步）
ORNOT H5.15  ; 腔体模式（0-正压 1-负压）
ANDLD
ANDNOT P_On
ORLD
LD D1075.06  ; #1腔体机构开腔体破真空阀/开电池破真空阀/开腔体阀（清氦步）
ANDNOT D1070.11  ; #1腔体机构关闭#1-1腔体阀/清氦判定（自动单检步）
ORLD
ANDLD
OUT 501.13  ; #1-1腔体阀开条件
LD TR0
LD 501.13  ; #1-1腔体阀开条件
OR 601.13  ; #1-1腔体阀开[A]
ANDLD
ANDNOT 821.00  ; #1-1腔体阀开到位标志
ANDNOT 511.13  ; #1-1腔体阀关条件
OUT 601.13  ; #1-1腔体阀开[A]
LD TR0
LD D1066.06  ; #1腔体机构关电池抽气阀（自动步）
AND H26.00  ; #1-1电池泄漏
LD D1066.07  ; #1腔体机构开电池注氦阀（自动步）
AND H26.02  ; #1-1电池注氦超时
ORLD
LD D1070.11  ; #1腔体机构关闭#1-1腔体阀/清氦判定（自动单检步）
ANDNOT H27.00  ; #1腔体有清氦需求
ORLD
LD D1074.04  ; #1腔体机构正压开腔体阀/负压关腔体阀/氦检阀打开
LD D1067.01  ; #1腔体机构清氦需求判定（自动步）
OR P_On
ANDLD
AND H5.15  ; 腔体模式（0-正压 1-负压）
ORLD
LD D1066.05  ; #1腔体机构腔体抽气阀打开/延时开电池抽气阀（自动步）  // #1-1无料时不测试
ANDNOT H25.00  ; #1-1腔体有料记忆
ORLD
ANDLD
OUT 511.13  ; #1-1腔体阀关条件
LD TR0
LD 511.13  ; #1-1腔体阀关条件
OR 611.13  ; #1-1腔体阀关[A]
ANDLD
ANDNOT 821.01  ; #1-1腔体阀关到位标志
ANDNOT 501.13  ; #1-1腔体阀开条件
OUT 611.13  ; #1-1腔体阀关[A]

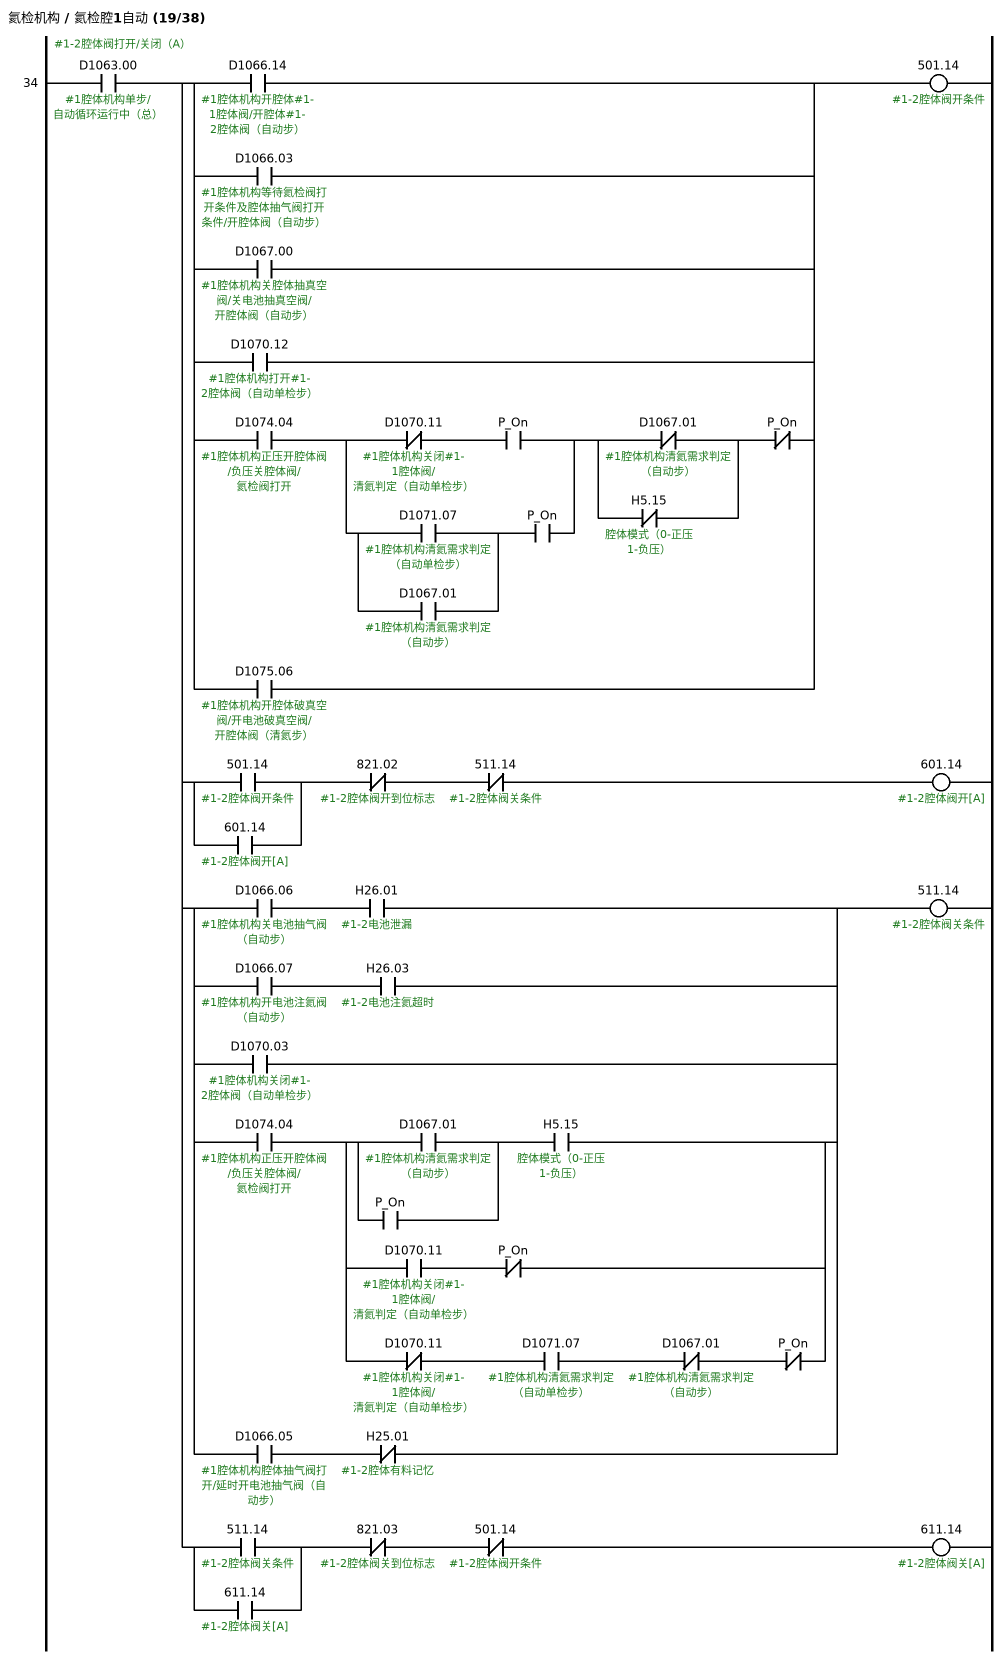
; rung 34: #1-2腔体阀打开/关闭（A）
LD D1063.00  ; #1腔体机构单步/自动循环运行中（总）
OUT TR0
LD D1066.14  ; #1腔体机构开腔体#1-1腔体阀/开腔体#1-2腔体阀（自动步）
OR D1066.03  ; #1腔体机构等待氦检阀打开条件及腔体抽气阀打开条件/开腔体阀（自动步）
OR D1067.00  ; #1腔体机构关腔体抽真空阀/关电池抽真空阀/开腔体阀（自动步）
OR D1070.12  ; #1腔体机构打开#1-2腔体阀（自动单检步）
LD D1074.04  ; #1腔体机构正压开腔体阀/负压关腔体阀/氦检阀打开
LDNOT D1070.11  ; #1腔体机构关闭#1-1腔体阀/清氦判定（自动单检步）
AND P_On
LD D1071.07  ; #1腔体机构清氦需求判定（自动单检步）
OR D1067.01  ; #1腔体机构清氦需求判定（自动步）
AND P_On
ORLD
ANDLD
LDNOT D1067.01  ; #1腔体机构清氦需求判定（自动步）
ORNOT H5.15  ; 腔体模式（0-正压 1-负压）
ANDLD
ANDNOT P_On
ORLD
OR D1075.06  ; #1腔体机构开腔体破真空阀/开电池破真空阀/开腔体阀（清氦步）
ANDLD
OUT 501.14  ; #1-2腔体阀开条件
LD TR0
LD 501.14  ; #1-2腔体阀开条件
OR 601.14  ; #1-2腔体阀开[A]
ANDLD
ANDNOT 821.02  ; #1-2腔体阀开到位标志
ANDNOT 511.14  ; #1-2腔体阀关条件
OUT 601.14  ; #1-2腔体阀开[A]
LD TR0
LD D1066.06  ; #1腔体机构关电池抽气阀（自动步）
AND H26.01  ; #1-2电池泄漏
LD D1066.07  ; #1腔体机构开电池注氦阀（自动步）
AND H26.03  ; #1-2电池注氦超时
ORLD
OR D1070.03  ; #1腔体机构关闭#1-2腔体阀（自动单检步）
LD D1074.04  ; #1腔体机构正压开腔体阀/负压关腔体阀/氦检阀打开
LD D1067.01  ; #1腔体机构清氦需求判定（自动步）
OR P_On
AND H5.15  ; 腔体模式（0-正压 1-负压）
LD D1070.11  ; #1腔体机构关闭#1-1腔体阀/清氦判定（自动单检步）
ANDNOT P_On
ORLD
LDNOT D1070.11  ; #1腔体机构关闭#1-1腔体阀/清氦判定（自动单检步）
AND D1071.07  ; #1腔体机构清氦需求判定（自动单检步）
ANDNOT D1067.01  ; #1腔体机构清氦需求判定（自动步）
ANDNOT P_On
ORLD
ANDLD
ORLD
LD D1066.05  ; #1腔体机构腔体抽气阀打开/延时开电池抽气阀（自动步）  // #1-2无料时不测试
ANDNOT H25.01  ; #1-2腔体有料记忆
ORLD
ANDLD
OUT 511.14  ; #1-2腔体阀关条件
LD TR0
LD 511.14  ; #1-2腔体阀关条件
OR 611.14  ; #1-2腔体阀关[A]
ANDLD
ANDNOT 821.03  ; #1-2腔体阀关到位标志
ANDNOT 501.14  ; #1-2腔体阀开条件
OUT 611.14  ; #1-2腔体阀关[A]

